LIN {X 0,Y 361.879,Z 141.036,A -85,B 0,C 180,E1 -13085.765,E2 -13085.765} C_VEL
LIN {X 0,Y 361.87,Z 141.034,A -85,B 0,C 180,E1 -13089.027,E2 -13089.027} C_VEL
LIN {X 0,Y 361.837,Z 141.037,A -85,B 0,C 180,E1 -13092.829,E2 -13092.829} C_VEL
LIN {X 0,Y 361.82,Z 141.044,A -85,B 0,C 180,E1 -13095.947,E2 -13095.947} C_VEL
LIN {X 0,Y 361.838,Z 141.042,A -85,B 0,C 180,E1 -13099.245,E2 -13099.245} C_VEL
LIN {X 0,Y 361.865,Z 141.033,A -85,B 0,C 180,E1 -13102.778,E2 -13102.778} C_VEL
LIN {X 0,Y 361.857,Z 141.036,A -85,B 0,C 180,E1 -13105.72,E2 -13105.72} C_VEL
LIN {X 0,Y 361.867,Z 141.03,A -85,B 0,C 180,E1 -13109.672,E2 -13109.672} C_VEL
LIN {X 0,Y 361.866,Z 141.018,A -85,B 0,C 180,E1 -13113.469,E2 -13113.469} C_VEL
LIN {X 0,Y 361.885,Z 141.028,A -85,B 0,C 180,E1 -13117.145,E2 -13117.145} C_VEL
LIN {X 0,Y 361.908,Z 141.031,A -85,B 0,C 180,E1 -13120.724,E2 -13120.724} C_VEL
LIN {X 0,Y 361.947,Z 141.019,A -85,B 0,C 180,E1 -13124.227,E2 -13124.227} C_VEL
LIN {X 0,Y 362.004,Z 141.017,A -85,B 0,C 180,E1 -13126.528,E2 -13126.528} C_VEL
LIN {X 0,Y 362.004,Z 141.016,A -85,B 0,C 180,E1 -13129.938,E2 -13129.938} C_VEL
LIN {X 0,Y 362.126,Z 140.997,A -85,B 0,C 180,E1 -13133.313,E2 -13133.313} C_VEL
LIN {X 0,Y 362.269,Z 140.97,A -85,B 0,C 180,E1 -13137.777,E2 -13137.777} C_VEL
LIN {X 0,Y 362.178,Z 140.979,A -85,B 0,C 180,E1 -13141.112,E2 -13141.112} C_VEL
LIN {X 0,Y 362.262,Z 140.976,A -85,B 0,C 180,E1 -13142.224,E2 -13142.224} C_VEL
LIN {X 0,Y 362.125,Z 140.992,A -85,B 0,C 180,E1 -13146.688,E2 -13146.688} C_VEL
LIN {X 0,Y 361.997,Z 140.99,A -85,B 0,C 180,E1 -13150.063,E2 -13150.063} C_VEL
LIN {X 0,Y 361.955,Z 141.024,A -85,B 0,C 180,E1 -13153.868,E2 -13153.868} C_VEL
LIN {X 0,Y 361.88,Z 141.031,A -85,B 0,C 180,E1 -13158.104,E2 -13158.104} C_VEL
LIN {X 0,Y 361.824,Z 141.034,A -85,B 0,C 180,E1 -13161.658,E2 -13161.658} C_VEL
LIN {X 0,Y 361.864,Z 141.037,A -85,B 0,C 180,E1 -13165.295,E2 -13165.295} C_VEL
LIN {X 0,Y 361.841,Z 141.012,A -85,B 0,C 180,E1 -13169.068,E2 -13169.068} C_VEL
LIN {X 0,Y 361.842,Z 141.028,A -85,B 0,C 180,E1 -13171.63,E2 -13171.63} C_VEL
LIN {X 0,Y 361.874,Z 141.028,A -85,B 0,C 180,E1 -13175.344,E2 -13175.344} C_VEL
LIN {X 0,Y 361.83,Z 141.018,A -85,B 0,C 180,E1 -13179.018,E2 -13179.018} C_VEL
LIN {X 0,Y 361.837,Z 141.039,A -85,B 0,C 180,E1 -13182.83,E2 -13182.83} C_VEL
LIN {X 0,Y 361.817,Z 141.02,A -85,B 0,C 180,E1 -13185.948,E2 -13185.948} C_VEL
LIN {X 0,Y 361.817,Z 141.04,A -85,B 0,C 180,E1 -13189.249,E2 -13189.249} C_VEL
LIN {X 0,Y 361.869,Z 141.025,A -85,B 0,C 180,E1 -13192.981,E2 -13192.981} C_VEL
LIN {X 0,Y 361.863,Z 141.027,A -85,B 0,C 180,E1 -13196.631,E2 -13196.631} C_VEL
LIN {X 0,Y 361.869,Z 141.035,A -85,B 0,C 180,E1 -13199.671,E2 -13199.671} C_VEL
LIN {X 0,Y 361.866,Z 141.036,A -85,B 0,C 180,E1 -13203.468,E2 -13203.468} C_VEL
LIN {X 0,Y 361.881,Z 141.033,A -85,B 0,C 180,E1 -13207.144,E2 -13207.144} C_VEL
LIN {X 0,Y 361.91,Z 141.025,A -85,B 0,C 180,E1 -13210.723,E2 -13210.723} C_VEL
LIN {X 0,Y 361.949,Z 141.027,A -85,B 0,C 180,E1 -13214.226,E2 -13214.226} C_VEL
LIN {X 0,Y 362.054,Z 141.133,A -85,B 0,C 180,E1 -13216.851,E2 -13216.851} C_VEL
LIN {X 0,Y 363.353,Z 146.545,A -85,B 0,C 180,E1 -13218.193,E2 -13218.193} C_VEL
LIN {X 0,Y 375.34,Z 174.664,A -85,B 0,C 180,E1 -13219.747,E2 -13219.747} C_VEL
LIN {X 0,Y 378.121,Z 181.605,A -85,B 0,C 180,E1 -13220.098,E2 -13220.098} C_VEL
LIN {X 0,Y 375.096,Z 311.282,A -85,B 0,C 180,E1 -13222.632,E2 -13222.632} C_VEL
LIN {X 0,Y 374.339,Z 326.412,A -85,B 0,C 180,E1 -13223.126,E2 -13223.126} C_VEL
LIN {X 0,Y 373.39,Z 340.483,A -85,B 0,C 180,E1 -13223.786,E2 -13223.786} C_VEL
LIN {X 0,Y 372.032,Z 355.504,A -85,B 0,C 180,E1 -13224.716,E2 -13224.716} C_VEL
LIN {X 0,Y 370.487,Z 370.541,A -85,B 0,C 180,E1 -13225.92,E2 -13225.92} C_VEL
LIN {X 0,Y 368.913,Z 383.973,A -85,B 0,C 180,E1 -13227.27,E2 -13227.27} C_VEL
LIN {X 0,Y 367.303,Z 396.209,A -85,B 0,C 180,E1 -13228.766,E2 -13228.766} C_VEL
LIN {X 0,Y 365.757,Z 407.68,A -85,B 0,C 180,E1 -13230.463,E2 -13230.463} C_VEL
LIN {X 0,Y 364.415,Z 417.514,A -85,B 0,C 180,E1 -13232.21,E2 -13232.21} C_VEL
LIN {X 0,Y 363.177,Z 426.655,A -85,B 0,C 180,E1 -13234.161,E2 -13234.161} C_VEL
LIN {X 0,Y 362.184,Z 434.264,A -85,B 0,C 180,E1 -13236.126,E2 -13236.126} C_VEL
LIN {X 0,Y 361.397,Z 441.384,A -85,B 0,C 180,E1 -13238.386,E2 -13238.386} C_VEL
LIN {X 0,Y 360.833,Z 447.004,A -85,B 0,C 180,E1 -13240.663,E2 -13240.663} C_VEL
LIN {X 0,Y 360.483,Z 451.14,A -85,B 0,C 180,E1 -13242.886,E2 -13242.886} C_VEL
LIN {X 0,Y 360.363,Z 452,A -85,B 0,C 180,E1 -13243.441,E2 -13243.441} C_VEL
LIN {X 0,Y 359.56,Z 453.289,A -85,B 0,C 180,E1 -13244.349,E2 -13244.349} C_VEL
LIN {X 0,Y 356.571,Z 454.897,A -85,B 0,C 180,E1 -13245.84,E2 -13245.84} C_VEL
LIN {X 0,Y 354.114,Z 455.843,A -85,B 0,C 180,E1 -13247.056,E2 -13247.056} C_VEL
LIN {X 0,Y 353.072,Z 456.303,A -85,B 0,C 180,E1 -13248.002,E2 -13248.002} C_VEL
LIN {X 0,Y 352.99,Z 456.411,A -85,B 0,C 180,E1 -13248.323,E2 -13248.323} C_VEL
LIN {X 0,Y 353.05,Z 456.561,A -85,B 0,C 180,E1 -13250.672,E2 -13250.672} C_VEL
LIN {X 0,Y 353.093,Z 456.028,A -85,B 0,C 180,E1 -13252.22,E2 -13252.22} C_VEL
LIN {X 0,Y 353.38,Z 454.051,A -85,B 0,C 180,E1 -13254.686,E2 -13254.686} C_VEL
LIN {X 0,Y 353.883,Z 450.673,A -85,B 0,C 180,E1 -13257.179,E2 -13257.179} C_VEL
LIN {X 0,Y 354.563,Z 445.772,A -85,B 0,C 180,E1 -13259.705,E2 -13259.705} C_VEL
LIN {X 0,Y 355.465,Z 440.501,A -85,B 0,C 180,E1 -13261.769,E2 -13261.769} C_VEL
LIN {X 0,Y 356.649,Z 433.956,A -85,B 0,C 180,E1 -13263.851,E2 -13263.851} C_VEL
LIN {X 0,Y 358.232,Z 425.446,A -85,B 0,C 180,E1 -13266.054,E2 -13266.054} C_VEL
LIN {X 0,Y 359.929,Z 416.53,A -85,B 0,C 180,E1 -13267.957,E2 -13267.957} C_VEL
LIN {X 0,Y 361.991,Z 405.841,A -85,B 0,C 180,E1 -13269.843,E2 -13269.843} C_VEL
LIN {X 0,Y 364.144,Z 394.025,A -85,B 0,C 180,E1 -13271.562,E2 -13271.562} C_VEL
LIN {X 0,Y 366.27,Z 381.307,A -85,B 0,C 180,E1 -13273.084,E2 -13273.084} C_VEL
LIN {X 0,Y 368.307,Z 368.431,A -85,B 0,C 180,E1 -13274.336,E2 -13274.336} C_VEL
LIN {X 0,Y 370.11,Z 354.336,A -85,B 0,C 180,E1 -13275.449,E2 -13275.449} C_VEL
LIN {X 0,Y 371.675,Z 340.065,A -85,B 0,C 180,E1 -13276.325,E2 -13276.325} C_VEL
LIN {X 0,Y 372.943,Z 325.224,A -85,B 0,C 180,E1 -13277.004,E2 -13277.004} C_VEL
LIN {X 0,Y 373.866,Z 310.283,A -85,B 0,C 180,E1 -13277.471,E2 -13277.471} C_VEL
LIN {X 0,Y 377.59,Z 188.012,A -85,B 0,C 180,E1 -13279.939,E2 -13279.939} C_VEL
LIN {X 0,Y 370.299,Z 172.503,A -85,B 0,C 180,E1 -13281.122,E2 -13281.122} C_VEL
LIN {X 0,Y 363.13,Z 159.246,A -85,B 0,C 180,E1 -13282.304,E2 -13282.304} C_VEL
LIN {X 0,Y 356.546,Z 147.757,A -85,B 0,C 180,E1 -13283.484,E2 -13283.484} C_VEL
LIN {X 0,Y 354.8,Z 141.906,A -85,B 0,C 180,E1 -13285.371,E2 -13285.371} C_VEL
LIN {X 0,Y 354.798,Z 141.908,A -85,B 0,C 180,E1 -13289.001,E2 -13289.001} C_VEL
LIN {X 0,Y 354.811,Z 141.899,A -85,B 0,C 180,E1 -13291.615,E2 -13291.615} C_VEL
LIN {X 0,Y 354.854,Z 141.892,A -85,B 0,C 180,E1 -13295.423,E2 -13295.423} C_VEL
LIN {X 0,Y 354.827,Z 141.91,A -85,B 0,C 180,E1 -13299.113,E2 -13299.113} C_VEL
LIN {X 0,Y 354.88,Z 141.902,A -85,B 0,C 180,E1 -13302.718,E2 -13302.718} C_VEL
LIN {X 0,Y 354.952,Z 141.897,A -85,B 0,C 180,E1 -13306.255,E2 -13306.255} C_VEL
LIN {X 0,Y 354.978,Z 141.894,A -85,B 0,C 180,E1 -13309.735,E2 -13309.735} C_VEL
LIN {X 0,Y 355.114,Z 141.874,A -85,B 0,C 180,E1 -13312.036,E2 -13312.036} C_VEL
LIN {X 0,Y 355.091,Z 141.87,A -85,B 0,C 180,E1 -13314.32,E2 -13314.32} C_VEL
LIN {X 0,Y 355.243,Z 141.853,A -85,B 0,C 180,E1 -13317.732,E2 -13317.732} C_VEL
LIN {X 0,Y 355.396,Z 141.84,A -85,B 0,C 180,E1 -13320,E2 -13320} C_VEL
LIN {X 0,Y 355.243,Z 141.855,A -85,B 0,C 180,E1 -13322.267,E2 -13322.267} C_VEL
LIN {X 0,Y 355.098,Z 141.877,A -85,B 0,C 180,E1 -13326.82,E2 -13326.82} C_VEL
LIN {X 0,Y 354.955,Z 141.893,A -85,B 0,C 180,E1 -13330.264,E2 -13330.264} C_VEL
LIN {X 0,Y 354.942,Z 141.896,A -85,B 0,C 180,E1 -13334.019,E2 -13334.019} C_VEL
LIN {X 0,Y 354.922,Z 141.899,A -85,B 0,C 180,E1 -13338.108,E2 -13338.108} C_VEL
LIN {X 0,Y 354.833,Z 141.909,A -85,B 0,C 180,E1 -13342.106,E2 -13342.106} C_VEL
LIN {X 0,Y 354.898,Z 141.898,A -85,B 0,C 180,E1 -13345.827,E2 -13345.827} C_VEL
LIN {X 0,Y 354.852,Z 141.903,A -85,B 0,C 180,E1 -13349.678,E2 -13349.678} C_VEL
LIN {X 0,Y 354.804,Z 141.914,A -85,B 0,C 180,E1 -13353.702,E2 -13353.702} C_VEL
LIN {X 0,Y 354.796,Z 141.917,A -85,B 0,C 180,E1 -13356.459,E2 -13356.459} C_VEL
LIN {X 0,Y 354.822,Z 141.896,A -85,B 0,C 180,E1 -13359.424,E2 -13359.424} C_VEL
LIN {X 0,Y 354.786,Z 141.901,A -85,B 0,C 180,E1 -13362.867,E2 -13362.867} C_VEL
LIN {X 0,Y 354.772,Z 141.909,A -85,B 0,C 180,E1 -13366.105,E2 -13366.105} C_VEL
LIN {X 0,Y 354.786,Z 141.911,A -85,B 0,C 180,E1 -13369.179,E2 -13369.179} C_VEL
LIN {X 0,Y 354.826,Z 141.959,A -85,B 0,C 180,E1 -13370.255,E2 -13370.255} C_VEL
LIN {X 0,Y 358.279,Z 153.223,A -85,B 0,C 180,E1 -13373.538,E2 -13373.538} C_VEL
LIN {X 0,Y 361.019,Z 163.125,A -85,B 0,C 180,E1 -13376.189,E2 -13376.189} C_VEL
LIN {X 0,Y 370.165,Z 181.186,A -85,B 0,C 180,E1 -13377.73,E2 -13377.73} C_VEL
LIN {X 0,Y 373.149,Z 188.13,A -85,B 0,C 180,E1 -13378.235,E2 -13378.235} C_VEL
LIN {X 0,Y 376.818,Z 207.275,A -85,B 0,C 180,E1 -13379.086,E2 -13379.086} C_VEL
LIN {X 0,Y 377.102,Z 209.697,A -85,B 0,C 180,E1 -13379.173,E2 -13379.173} C_VEL
LIN {X 0,Y 373.367,Z 329.597,A -85,B 0,C 180,E1 -13381.584,E2 -13381.584} C_VEL
LIN {X 0,Y 372.224,Z 345.584,A -85,B 0,C 180,E1 -13382.103,E2 -13382.103} C_VEL
LIN {X 0,Y 370.742,Z 360.136,A -85,B 0,C 180,E1 -13382.786,E2 -13382.786} C_VEL
LIN {X 0,Y 368.921,Z 374.936,A -85,B 0,C 180,E1 -13383.717,E2 -13383.717} C_VEL
LIN {X 0,Y 367.076,Z 388.167,A -85,B 0,C 180,E1 -13384.787,E2 -13384.787} C_VEL
LIN {X 0,Y 364.789,Z 401.788,A -85,B 0,C 180,E1 -13386.135,E2 -13386.135} C_VEL
LIN {X 0,Y 362.674,Z 414.145,A -85,B 0,C 180,E1 -13387.648,E2 -13387.648} C_VEL
LIN {X 0,Y 360.496,Z 425.702,A -85,B 0,C 180,E1 -13389.353,E2 -13389.353} C_VEL
LIN {X 0,Y 358.711,Z 435.703,A -85,B 0,C 180,E1 -13391.139,E2 -13391.139} C_VEL
LIN {X 0,Y 357.011,Z 444.998,A -85,B 0,C 180,E1 -13393.121,E2 -13393.121} C_VEL
LIN {X 0,Y 355.666,Z 452.763,A -85,B 0,C 180,E1 -13395.115,E2 -13395.115} C_VEL
LIN {X 0,Y 354.777,Z 458.414,A -85,B 0,C 180,E1 -13396.832,E2 -13396.832} C_VEL
LIN {X 0,Y 353.955,Z 464.549,A -85,B 0,C 180,E1 -13399.128,E2 -13399.128} C_VEL
LIN {X 0,Y 353.498,Z 469.304,A -85,B 0,C 180,E1 -13401.425,E2 -13401.425} C_VEL
LIN {X 0,Y 353.275,Z 473.279,A -85,B 0,C 180,E1 -13404.092,E2 -13404.092} C_VEL
LIN {X 0,Y 353.19,Z 475.51,A -85,B 0,C 180,E1 -13406.578,E2 -13406.578} C_VEL
LIN {X 0,Y 353.211,Z 476.343,A -85,B 0,C 180,E1 -13408.86,E2 -13408.86} C_VEL
LIN {X 0,Y 353.215,Z 476.037,A -85,B 0,C 180,E1 -13411.141,E2 -13411.141} C_VEL
LIN {X 0,Y 353.194,Z 474.577,A -85,B 0,C 180,E1 -13413.423,E2 -13413.423} C_VEL
LIN {X 0,Y 353.275,Z 471.617,A -85,B 0,C 180,E1 -13415.909,E2 -13415.909} C_VEL
LIN {X 0,Y 353.427,Z 467.984,A -85,B 0,C 180,E1 -13418.002,E2 -13418.002} C_VEL
LIN {X 0,Y 353.698,Z 462.674,A -85,B 0,C 180,E1 -13420.302,E2 -13420.302} C_VEL
LIN {X 0,Y 354.396,Z 455.88,A -85,B 0,C 180,E1 -13422.6,E2 -13422.6} C_VEL
LIN {X 0,Y 355.211,Z 448.529,A -85,B 0,C 180,E1 -13424.613,E2 -13424.613} C_VEL
LIN {X 0,Y 356.304,Z 439.69,A -85,B 0,C 180,E1 -13426.62,E2 -13426.62} C_VEL
LIN {X 0,Y 357.857,Z 429.042,A -85,B 0,C 180,E1 -13428.611,E2 -13428.611} C_VEL
LIN {X 0,Y 359.237,Z 418.762,A -85,B 0,C 180,E1 -13430.217,E2 -13430.217} C_VEL
LIN {X 0,Y 360.81,Z 407.288,A -85,B 0,C 180,E1 -13431.722,E2 -13431.722} C_VEL
LIN {X 0,Y 362.485,Z 394.416,A -85,B 0,C 180,E1 -13433.118,E2 -13433.118} C_VEL
LIN {X 0,Y 364.026,Z 382.022,A -85,B 0,C 180,E1 -13434.222,E2 -13434.222} C_VEL
LIN {X 0,Y 365.576,Z 367.655,A -85,B 0,C 180,E1 -13435.248,E2 -13435.248} C_VEL
LIN {X 0,Y 366.71,Z 353.667,A -85,B 0,C 180,E1 -13436.031,E2 -13436.031} C_VEL
LIN {X 0,Y 367.849,Z 338.418,A -85,B 0,C 180,E1 -13436.641,E2 -13436.641} C_VEL
LIN {X 0,Y 368.459,Z 322.812,A -85,B 0,C 180,E1 -13437.052,E2 -13437.052} C_VEL
LIN {X 0,Y 371.276,Z 207.418,A -85,B 0,C 180,E1 -13439.317,E2 -13439.317} C_VEL
LIN {X 0,Y 365.889,Z 177.835,A -85,B 0,C 180,E1 -13440.363,E2 -13440.363} C_VEL
LIN {X 0,Y 360.228,Z 163.937,A -85,B 0,C 180,E1 -13441.146,E2 -13441.146} C_VEL
LIN {X 0,Y 356.983,Z 150.277,A -85,B 0,C 180,E1 -13444.223,E2 -13444.223} C_VEL
LIN {X 0,Y 354.838,Z 141.912,A -85,B 0,C 180,E1 -13446.245,E2 -13446.245} C_VEL
LIN {X 0,Y 354.825,Z 141.914,A -85,B 0,C 180,E1 -13449.424,E2 -13449.424} C_VEL
LIN {X 0,Y 354.789,Z 141.916,A -85,B 0,C 180,E1 -13452.868,E2 -13452.868} C_VEL
LIN {X 0,Y 354.769,Z 141.922,A -85,B 0,C 180,E1 -13456.104,E2 -13456.104} C_VEL
LIN {X 0,Y 354.79,Z 141.921,A -85,B 0,C 180,E1 -13459.18,E2 -13459.18} C_VEL
LIN {X 0,Y 354.808,Z 141.911,A -85,B 0,C 180,E1 -13462.403,E2 -13462.403} C_VEL
LIN {X 0,Y 354.814,Z 141.911,A -85,B 0,C 180,E1 -13464.941,E2 -13464.941} C_VEL
LIN {X 0,Y 354.796,Z 141.913,A -85,B 0,C 180,E1 -13468.406,E2 -13468.406} C_VEL
LIN {X 0,Y 354.802,Z 141.894,A -85,B 0,C 180,E1 -13471.615,E2 -13471.615} C_VEL
LIN {X 0,Y 354.838,Z 141.907,A -85,B 0,C 180,E1 -13475.658,E2 -13475.658} C_VEL
LIN {X 0,Y 354.83,Z 141.907,A -85,B 0,C 180,E1 -13479.114,E2 -13479.114} C_VEL
LIN {X 0,Y 354.884,Z 141.898,A -85,B 0,C 180,E1 -13482.72,E2 -13482.72} C_VEL
LIN {X 0,Y 354.956,Z 141.896,A -85,B 0,C 180,E1 -13486.256,E2 -13486.256} C_VEL
LIN {X 0,Y 354.96,Z 141.892,A -85,B 0,C 180,E1 -13489.736,E2 -13489.736} C_VEL
LIN {X 0,Y 355.092,Z 141.874,A -85,B 0,C 180,E1 -13493.18,E2 -13493.18} C_VEL
LIN {X 0,Y 355.231,Z 141.847,A -85,B 0,C 180,E1 -13497.733,E2 -13497.733} C_VEL
LIN {X 0,Y 355.149,Z 141.854,A -85,B 0,C 180,E1 -13501.134,E2 -13501.134} C_VEL
LIN {X 0,Y 355.224,Z 141.853,A -85,B 0,C 180,E1 -13502.268,E2 -13502.268} C_VEL
LIN {X 0,Y 355.092,Z 141.867,A -85,B 0,C 180,E1 -13506.821,E2 -13506.821} C_VEL
LIN {X 0,Y 354.953,Z 141.868,A -85,B 0,C 180,E1 -13510.265,E2 -13510.265} C_VEL
LIN {X 0,Y 354.897,Z 141.903,A -85,B 0,C 180,E1 -13513.986,E2 -13513.986} C_VEL
LIN {X 0,Y 354.837,Z 141.908,A -85,B 0,C 180,E1 -13518.064,E2 -13518.064} C_VEL
LIN {X 0,Y 354.791,Z 141.909,A -85,B 0,C 180,E1 -13522.109,E2 -13522.109} C_VEL
LIN {X 0,Y 354.803,Z 141.91,A -85,B 0,C 180,E1 -13525.836,E2 -13525.836} C_VEL
LIN {X 0,Y 354.79,Z 141.889,A -85,B 0,C 180,E1 -13529.685,E2 -13529.685} C_VEL
LIN {X 0,Y 354.791,Z 141.908,A -85,B 0,C 180,E1 -13532.334,E2 -13532.334} C_VEL
LIN {X 0,Y 354.823,Z 141.904,A -85,B 0,C 180,E1 -13535.698,E2 -13535.698} C_VEL
LIN {X 0,Y 354.773,Z 141.901,A -85,B 0,C 180,E1 -13539.413,E2 -13539.413} C_VEL
LIN {X 0,Y 354.789,Z 141.916,A -85,B 0,C 180,E1 -13542.866,E2 -13542.866} C_VEL
LIN {X 0,Y 354.767,Z 141.898,A -85,B 0,C 180,E1 -13546.103,E2 -13546.103} C_VEL
LIN {X 0,Y 354.77,Z 141.918,A -85,B 0,C 180,E1 -13549.176,E2 -13549.176} C_VEL
LIN {X 0,Y 354.805,Z 141.901,A -85,B 0,C 180,E1 -13552.404,E2 -13552.404} C_VEL
LIN {X 0,Y 354.816,Z 141.913,A -85,B 0,C 180,E1 -13554.941,E2 -13554.941} C_VEL
LIN {X 0,Y 354.798,Z 141.91,A -85,B 0,C 180,E1 -13558.405,E2 -13558.405} C_VEL
LIN {X 0,Y 354.804,Z 141.909,A -85,B 0,C 180,E1 -13561.614,E2 -13561.614} C_VEL
LIN {X 0,Y 354.811,Z 141.915,A -85,B 0,C 180,E1 -13565.419,E2 -13565.419} C_VEL
LIN {X 0,Y 354.832,Z 141.91,A -85,B 0,C 180,E1 -13569.113,E2 -13569.113} C_VEL
LIN {X 0,Y 354.885,Z 141.887,A -85,B 0,C 180,E1 -13572.719,E2 -13572.719} C_VEL
LIN {X 0,Y 355,Z 142.038,A -85,B 0,C 180,E1 -13576.402,E2 -13576.402} C_VEL
LIN {X 0,Y 356.226,Z 147.086,A -85,B 0,C 180,E1 -13577.637,E2 -13577.637} C_VEL
LIN {X 0,Y 368.488,Z 175.376,A -85,B 0,C 180,E1 -13579.247,E2 -13579.247} C_VEL
LIN {X 0,Y 371.75,Z 183.518,A -85,B 0,C 180,E1 -13579.668,E2 -13579.668} C_VEL
LIN {X 0,Y 368.535,Z 312.21,A -85,B 0,C 180,E1 -13582.225,E2 -13582.225} C_VEL
LIN {X 0,Y 367.701,Z 327.89,A -85,B 0,C 180,E1 -13582.759,E2 -13582.759} C_VEL
LIN {X 0,Y 366.687,Z 342.3,A -85,B 0,C 180,E1 -13583.465,E2 -13583.465} C_VEL
LIN {X 0,Y 365.379,Z 355.987,A -85,B 0,C 180,E1 -13584.342,E2 -13584.342} C_VEL
LIN {X 0,Y 363.97,Z 369.407,A -85,B 0,C 180,E1 -13585.431,E2 -13585.431} C_VEL
LIN {X 0,Y 362.295,Z 383.114,A -85,B 0,C 180,E1 -13586.802,E2 -13586.802} C_VEL
LIN {X 0,Y 360.596,Z 395.529,A -85,B 0,C 180,E1 -13588.324,E2 -13588.324} C_VEL
LIN {X 0,Y 359.028,Z 406.818,A -85,B 0,C 180,E1 -13590,E2 -13590} C_VEL
LIN {X 0,Y 357.709,Z 416.331,A -85,B 0,C 180,E1 -13591.688,E2 -13591.688} C_VEL
LIN {X 0,Y 356.366,Z 425.713,A -85,B 0,C 180,E1 -13593.674,E2 -13593.674} C_VEL
LIN {X 0,Y 355.302,Z 433.529,A -85,B 0,C 180,E1 -13595.675,E2 -13595.675} C_VEL
LIN {X 0,Y 354.452,Z 440.836,A -85,B 0,C 180,E1 -13597.978,E2 -13597.978} C_VEL
LIN {X 0,Y 353.797,Z 446.631,A -85,B 0,C 180,E1 -13600.298,E2 -13600.298} C_VEL
LIN {X 0,Y 353.438,Z 451.033,A -85,B 0,C 180,E1 -13602.634,E2 -13602.634} C_VEL
LIN {X 0,Y 353.107,Z 454.159,A -85,B 0,C 180,E1 -13604.995,E2 -13604.995} C_VEL
LIN {X 0,Y 353.039,Z 456.034,A -85,B 0,C 180,E1 -13607.374,E2 -13607.374} C_VEL
LIN {X 0,Y 352.99,Z 456.411,A -85,B 0,C 180,E1 -13608.323,E2 -13608.323} C_VEL
LIN {X 0,Y 352.321,Z 456.687,A -85,B 0,C 180,E1 -13609.275,E2 -13609.275} C_VEL
LIN {X 0,Y 349.461,Z 456.693,A -85,B 0,C 180,E1 -13610.826,E2 -13610.826} C_VEL
LIN {X 0,Y 347.091,Z 456.3,A -85,B 0,C 180,E1 -13612.081,E2 -13612.081} C_VEL
LIN {X 0,Y 346.146,Z 455.783,A -85,B 0,C 180,E1 -13613.048,E2 -13613.048} C_VEL
LIN {X 0,Y 346.108,Z 455.534,A -85,B 0,C 180,E1 -13613.374,E2 -13613.374} C_VEL
LIN {X 0,Y 346.372,Z 453.872,A -85,B 0,C 180,E1 -13615.22,E2 -13615.22} C_VEL
LIN {X 0,Y 346.917,Z 450.294,A -85,B 0,C 180,E1 -13617.771,E2 -13617.771} C_VEL
LIN {X 0,Y 347.737,Z 445.156,A -85,B 0,C 180,E1 -13620.349,E2 -13620.349} C_VEL
LIN {X 0,Y 348.765,Z 439.682,A -85,B 0,C 180,E1 -13622.477,E2 -13622.477} C_VEL
LIN {X 0,Y 350.086,Z 432.868,A -85,B 0,C 180,E1 -13624.605,E2 -13624.605} C_VEL
LIN {X 0,Y 351.867,Z 424.207,A -85,B 0,C 180,E1 -13626.813,E2 -13626.813} C_VEL
LIN {X 0,Y 353.658,Z 414.975,A -85,B 0,C 180,E1 -13628.754,E2 -13628.754} C_VEL
LIN {X 0,Y 355.894,Z 403.932,A -85,B 0,C 180,E1 -13630.667,E2 -13630.667} C_VEL
LIN {X 0,Y 358.205,Z 391.69,A -85,B 0,C 180,E1 -13632.41,E2 -13632.41} C_VEL
LIN {X 0,Y 360.301,Z 379.771,A -85,B 0,C 180,E1 -13633.803,E2 -13633.803} C_VEL
LIN {X 0,Y 362.397,Z 366.663,A -85,B 0,C 180,E1 -13635.06,E2 -13635.06} C_VEL
LIN {X 0,Y 364.223,Z 352.726,A -85,B 0,C 180,E1 -13636.142,E2 -13636.142} C_VEL
LIN {X 0,Y 365.803,Z 338.606,A -85,B 0,C 180,E1 -13636.991,E2 -13636.991} C_VEL
LIN {X 0,Y 367.041,Z 324.609,A -85,B 0,C 180,E1 -13637.62,E2 -13637.62} C_VEL
LIN {X 0,Y 367.904,Z 310.5,A -85,B 0,C 180,E1 -13638.066,E2 -13638.066} C_VEL
LIN {X 0,Y 371.748,Z 190.159,A -85,B 0,C 180,E1 -13640.529,E2 -13640.529} C_VEL
LIN {X 0,Y 364.564,Z 175.02,A -85,B 0,C 180,E1 -13641.734,E2 -13641.734} C_VEL
LIN {X 0,Y 356.643,Z 160.458,A -85,B 0,C 180,E1 -13643.1,E2 -13643.1} C_VEL
LIN {X 0,Y 351.183,Z 151.357,A -85,B 0,C 180,E1 -13644.077,E2 -13644.077} C_VEL
LIN {X 0,Y 349.378,Z 148.082,A -85,B 0,C 180,E1 -13644.445,E2 -13644.445} C_VEL
LIN {X 0,Y 347.773,Z 142.789,A -85,B 0,C 180,E1 -13646.234,E2 -13646.234} C_VEL
LIN {X 0,Y 347.745,Z 142.795,A -85,B 0,C 180,E1 -13649.651,E2 -13649.651} C_VEL
LIN {X 0,Y 347.785,Z 142.789,A -85,B 0,C 180,E1 -13653.603,E2 -13653.603} C_VEL
LIN {X 0,Y 347.784,Z 142.77,A -85,B 0,C 180,E1 -13656.161,E2 -13656.161} C_VEL
LIN {X 0,Y 347.806,Z 142.783,A -85,B 0,C 180,E1 -13659.908,E2 -13659.908} C_VEL
LIN {X 0,Y 347.832,Z 142.784,A -85,B 0,C 180,E1 -13663.568,E2 -13663.568} C_VEL
LIN {X 0,Y 347.89,Z 142.775,A -85,B 0,C 180,E1 -13667.16,E2 -13667.16} C_VEL
LIN {X 0,Y 348.094,Z 142.745,A -85,B 0,C 180,E1 -13671.612,E2 -13671.612} C_VEL
LIN {X 0,Y 348.066,Z 142.746,A -85,B 0,C 180,E1 -13674.205,E2 -13674.205} C_VEL
LIN {X 0,Y 348.205,Z 142.729,A -85,B 0,C 180,E1 -13677.686,E2 -13677.686} C_VEL
LIN {X 0,Y 348.345,Z 142.718,A -85,B 0,C 180,E1 -13680,E2 -13680} C_VEL
LIN {X 0,Y 348.206,Z 142.732,A -85,B 0,C 180,E1 -13682.313,E2 -13682.313} C_VEL
LIN {X 0,Y 348.063,Z 142.754,A -85,B 0,C 180,E1 -13686.958,E2 -13686.958} C_VEL
LIN {X 0,Y 347.896,Z 142.774,A -85,B 0,C 180,E1 -13690.475,E2 -13690.475} C_VEL
LIN {X 0,Y 347.897,Z 142.773,A -85,B 0,C 180,E1 -13694.149,E2 -13694.149} C_VEL
LIN {X 0,Y 347.89,Z 142.775,A -85,B 0,C 180,E1 -13698.29,E2 -13698.29} C_VEL
LIN {X 0,Y 347.787,Z 142.787,A -85,B 0,C 180,E1 -13701.635,E2 -13701.635} C_VEL
LIN {X 0,Y 347.811,Z 142.784,A -85,B 0,C 180,E1 -13705.108,E2 -13705.108} C_VEL
LIN {X 0,Y 347.809,Z 142.785,A -85,B 0,C 180,E1 -13707.694,E2 -13707.694} C_VEL
LIN {X 0,Y 347.762,Z 142.79,A -85,B 0,C 180,E1 -13710.346,E2 -13710.346} C_VEL
LIN {X 0,Y 347.742,Z 142.791,A -85,B 0,C 180,E1 -13714.464,E2 -13714.464} C_VEL
LIN {X 0,Y 347.771,Z 142.774,A -85,B 0,C 180,E1 -13717.988,E2 -13717.988} C_VEL
LIN {X 0,Y 347.748,Z 142.787,A -85,B 0,C 180,E1 -13721.83,E2 -13721.83} C_VEL
LIN {X 0,Y 347.764,Z 142.793,A -85,B 0,C 180,E1 -13725.017,E2 -13725.017} C_VEL
LIN {X 0,Y 347.761,Z 142.789,A -85,B 0,C 180,E1 -13728.944,E2 -13728.944} C_VEL
LIN {X 0,Y 347.761,Z 142.903,A -85,B 0,C 180,E1 -13729.391,E2 -13729.391} C_VEL
LIN {X 0,Y 351.251,Z 154.011,A -85,B 0,C 180,E1 -13732.774,E2 -13732.774} C_VEL
LIN {X 0,Y 353.862,Z 163.089,A -85,B 0,C 180,E1 -13735.258,E2 -13735.258} C_VEL
LIN {X 0,Y 363.123,Z 180.892,A -85,B 0,C 180,E1 -13736.895,E2 -13736.895} C_VEL
LIN {X 0,Y 367.729,Z 191.04,A -85,B 0,C 180,E1 -13737.69,E2 -13737.69} C_VEL
LIN {X 0,Y 371.148,Z 209.403,A -85,B 0,C 180,E1 -13738.521,E2 -13738.521} C_VEL
LIN {X 0,Y 369.725,Z 257.449,A -85,B 0,C 180,E1 -13739.508,E2 -13739.508} C_VEL
LIN {X 0,Y 367.386,Z 329.786,A -85,B 0,C 180,E1 -13741,E2 -13741} C_VEL
LIN {X 0,Y 366.183,Z 345.589,A -85,B 0,C 180,E1 -13741.523,E2 -13741.523} C_VEL
LIN {X 0,Y 364.64,Z 360.075,A -85,B 0,C 180,E1 -13742.213,E2 -13742.213} C_VEL
LIN {X 0,Y 362.755,Z 374.729,A -85,B 0,C 180,E1 -13743.15,E2 -13743.15} C_VEL
LIN {X 0,Y 360.706,Z 388.806,A -85,B 0,C 180,E1 -13744.309,E2 -13744.309} C_VEL
LIN {X 0,Y 358.333,Z 402.268,A -85,B 0,C 180,E1 -13745.678,E2 -13745.678} C_VEL
LIN {X 0,Y 355.919,Z 415.512,A -85,B 0,C 180,E1 -13747.354,E2 -13747.354} C_VEL
LIN {X 0,Y 353.728,Z 426.576,A -85,B 0,C 180,E1 -13749.046,E2 -13749.046} C_VEL
LIN {X 0,Y 351.695,Z 437.341,A -85,B 0,C 180,E1 -13751.051,E2 -13751.051} C_VEL
LIN {X 0,Y 349.963,Z 446.338,A -85,B 0,C 180,E1 -13753.071,E2 -13753.071} C_VEL
LIN {X 0,Y 348.371,Z 454.744,A -85,B 0,C 180,E1 -13755.374,E2 -13755.374} C_VEL
LIN {X 0,Y 347.399,Z 461.649,A -85,B 0,C 180,E1 -13757.736,E2 -13757.736} C_VEL
LIN {X 0,Y 346.643,Z 467.04,A -85,B 0,C 180,E1 -13760.077,E2 -13760.077} C_VEL
LIN {X 0,Y 346.366,Z 470.203,A -85,B 0,C 180,E1 -13761.835,E2 -13761.835} C_VEL
LIN {X 0,Y 346.158,Z 473.387,A -85,B 0,C 180,E1 -13764.174,E2 -13764.174} C_VEL
LIN {X 0,Y 346.112,Z 475.359,A -85,B 0,C 180,E1 -13766.508,E2 -13766.508} C_VEL
LIN {X 0,Y 346.111,Z 476.152,A -85,B 0,C 180,E1 -13768.837,E2 -13768.837} C_VEL
LIN {X 0,Y 346.115,Z 475.808,A -85,B 0,C 180,E1 -13771.164,E2 -13771.164} C_VEL
LIN {X 0,Y 346.117,Z 474.31,A -85,B 0,C 180,E1 -13773.493,E2 -13773.493} C_VEL
LIN {X 0,Y 346.195,Z 471.531,A -85,B 0,C 180,E1 -13775.885,E2 -13775.885} C_VEL
LIN {X 0,Y 346.35,Z 467.651,A -85,B 0,C 180,E1 -13778.166,E2 -13778.166} C_VEL
LIN {X 0,Y 346.656,Z 462.293,A -85,B 0,C 180,E1 -13780.514,E2 -13780.514} C_VEL
LIN {X 0,Y 347.398,Z 455.448,A -85,B 0,C 180,E1 -13782.858,E2 -13782.858} C_VEL
LIN {X 0,Y 348.245,Z 448.159,A -85,B 0,C 180,E1 -13784.881,E2 -13784.881} C_VEL
LIN {X 0,Y 349.422,Z 439.141,A -85,B 0,C 180,E1 -13786.957,E2 -13786.957} C_VEL
LIN {X 0,Y 351.044,Z 428.421,A -85,B 0,C 180,E1 -13788.986,E2 -13788.986} C_VEL
LIN {X 0,Y 352.574,Z 416.976,A -85,B 0,C 180,E1 -13790.782,E2 -13790.782} C_VEL
LIN {X 0,Y 354.32,Z 405.291,A -85,B 0,C 180,E1 -13792.294,E2 -13792.294} C_VEL
LIN {X 0,Y 356.03,Z 392.025,A -85,B 0,C 180,E1 -13793.716,E2 -13793.716} C_VEL
LIN {X 0,Y 357.701,Z 379.124,A -85,B 0,C 180,E1 -13794.833,E2 -13794.833} C_VEL
LIN {X 0,Y 359.238,Z 364.426,A -85,B 0,C 180,E1 -13795.852,E2 -13795.852} C_VEL
LIN {X 0,Y 360.493,Z 349.412,A -85,B 0,C 180,E1 -13796.642,E2 -13796.642} C_VEL
LIN {X 0,Y 361.522,Z 333.568,A -85,B 0,C 180,E1 -13797.223,E2 -13797.223} C_VEL
LIN {X 0,Y 362.268,Z 311.772,A -85,B 0,C 180,E1 -13797.71,E2 -13797.71} C_VEL
LIN {X 0,Y 364.858,Z 208.371,A -85,B 0,C 180,E1 -13799.773,E2 -13799.773} C_VEL
LIN {X 0,Y 359.888,Z 180.715,A -85,B 0,C 180,E1 -13800.769,E2 -13800.769} C_VEL
LIN {X 0,Y 352.97,Z 163.804,A -85,B 0,C 180,E1 -13801.733,E2 -13801.733} C_VEL
LIN {X 0,Y 349.987,Z 151.467,A -85,B 0,C 180,E1 -13804.583,E2 -13804.583} C_VEL
LIN {X 0,Y 347.786,Z 142.793,A -85,B 0,C 180,E1 -13806.698,E2 -13806.698} C_VEL
LIN {X 0,Y 347.733,Z 142.797,A -85,B 0,C 180,E1 -13810.298,E2 -13810.298} C_VEL
LIN {X 0,Y 347.724,Z 142.8,A -85,B 0,C 180,E1 -13813.409,E2 -13813.409} C_VEL
LIN {X 0,Y 347.727,Z 142.799,A -85,B 0,C 180,E1 -13816.687,E2 -13816.687} C_VEL
LIN {X 0,Y 347.749,Z 142.788,A -85,B 0,C 180,E1 -13820.174,E2 -13820.174} C_VEL
LIN {X 0,Y 347.763,Z 142.789,A -85,B 0,C 180,E1 -13822.68,E2 -13822.68} C_VEL
LIN {X 0,Y 347.751,Z 142.792,A -85,B 0,C 180,E1 -13825.957,E2 -13825.957} C_VEL
LIN {X 0,Y 347.743,Z 142.79,A -85,B 0,C 180,E1 -13829.652,E2 -13829.652} C_VEL
LIN {X 0,Y 347.752,Z 142.777,A -85,B 0,C 180,E1 -13833.602,E2 -13833.602} C_VEL
LIN {X 0,Y 347.778,Z 142.786,A -85,B 0,C 180,E1 -13836.162,E2 -13836.162} C_VEL
LIN {X 0,Y 347.809,Z 142.782,A -85,B 0,C 180,E1 -13839.91,E2 -13839.91} C_VEL
LIN {X 0,Y 347.836,Z 142.775,A -85,B 0,C 180,E1 -13843.569,E2 -13843.569} C_VEL
LIN {X 0,Y 347.894,Z 142.768,A -85,B 0,C 180,E1 -13847.161,E2 -13847.161} C_VEL
LIN {X 0,Y 347.939,Z 142.768,A -85,B 0,C 180,E1 -13850.701,E2 -13850.701} C_VEL
LIN {X 0,Y 348.043,Z 142.756,A -85,B 0,C 180,E1 -13854.206,E2 -13854.206} C_VEL
LIN {X 0,Y 348.192,Z 142.723,A -85,B 0,C 180,E1 -13857.687,E2 -13857.687} C_VEL
LIN {X 0,Y 348.121,Z 142.729,A -85,B 0,C 180,E1 -13861.157,E2 -13861.157} C_VEL
LIN {X 0,Y 348.185,Z 142.73,A -85,B 0,C 180,E1 -13862.314,E2 -13862.314} C_VEL
LIN {X 0,Y 348.059,Z 142.743,A -85,B 0,C 180,E1 -13866.959,E2 -13866.959} C_VEL
LIN {X 0,Y 347.892,Z 142.749,A -85,B 0,C 180,E1 -13870.476,E2 -13870.476} C_VEL
LIN {X 0,Y 347.856,Z 142.779,A -85,B 0,C 180,E1 -13874.119,E2 -13874.119} C_VEL
LIN {X 0,Y 347.79,Z 142.785,A -85,B 0,C 180,E1 -13878.237,E2 -13878.237} C_VEL
LIN {X 0,Y 347.748,Z 142.787,A -85,B 0,C 180,E1 -13881.616,E2 -13881.616} C_VEL
LIN {X 0,Y 347.741,Z 142.795,A -85,B 0,C 180,E1 -13885.114,E2 -13885.114} C_VEL
LIN {X 0,Y 347.729,Z 142.778,A -85,B 0,C 180,E1 -13887.702,E2 -13887.702} C_VEL
LIN {X 0,Y 347.737,Z 142.771,A -85,B 0,C 180,E1 -13890.35,E2 -13890.35} C_VEL
LIN {X 0,Y 347.753,Z 142.79,A -85,B 0,C 180,E1 -13894.044,E2 -13894.044} C_VEL
LIN {X 0,Y 347.759,Z 142.769,A -85,B 0,C 180,E1 -13897.322,E2 -13897.322} C_VEL
LIN {X 0,Y 347.746,Z 142.791,A -85,B 0,C 180,E1 -13901.601,E2 -13901.601} C_VEL
LIN {X 0,Y 347.704,Z 142.78,A -85,B 0,C 180,E1 -13905.028,E2 -13905.028} C_VEL
LIN {X 0,Y 347.746,Z 142.791,A -85,B 0,C 180,E1 -13908.399,E2 -13908.399} C_VEL
LIN {X 0,Y 347.761,Z 142.779,A -85,B 0,C 180,E1 -13912.678,E2 -13912.678} C_VEL
LIN {X 0,Y 347.754,Z 142.792,A -85,B 0,C 180,E1 -13915.956,E2 -13915.956} C_VEL
LIN {X 0,Y 347.746,Z 142.794,A -85,B 0,C 180,E1 -13919.651,E2 -13919.651} C_VEL
LIN {X 0,Y 347.749,Z 142.796,A -85,B 0,C 180,E1 -13923.6,E2 -13923.6} C_VEL
LIN {X 0,Y 347.757,Z 142.795,A -85,B 0,C 180,E1 -13926.159,E2 -13926.159} C_VEL
LIN {X 0,Y 347.811,Z 142.788,A -85,B 0,C 180,E1 -13929.909,E2 -13929.909} C_VEL
LIN {X 0,Y 347.837,Z 142.773,A -85,B 0,C 180,E1 -13933.568,E2 -13933.568} C_VEL
LIN {X 0,Y 347.909,Z 142.796,A -85,B 0,C 180,E1 -13935.906,E2 -13935.906} C_VEL
LIN {X 0,Y 348.94,Z 147.03,A -85,B 0,C 180,E1 -13937.005,E2 -13937.005} C_VEL
LIN {X 0,Y 361.391,Z 175.438,A -85,B 0,C 180,E1 -13938.697,E2 -13938.697} C_VEL
LIN {X 0,Y 365.326,Z 185.606,A -85,B 0,C 180,E1 -13939.229,E2 -13939.229} C_VEL
LIN {X 0,Y 362.066,Z 311.741,A -85,B 0,C 180,E1 -13941.769,E2 -13941.769} C_VEL
LIN {X 0,Y 361.201,Z 327.692,A -85,B 0,C 180,E1 -13942.312,E2 -13942.312} C_VEL
LIN {X 0,Y 360.19,Z 341.575,A -85,B 0,C 180,E1 -13942.995,E2 -13942.995} C_VEL
LIN {X 0,Y 358.756,Z 356.439,A -85,B 0,C 180,E1 -13943.955,E2 -13943.955} C_VEL
LIN {X 0,Y 357.287,Z 369.828,A -85,B 0,C 180,E1 -13945.063,E2 -13945.063} C_VEL
LIN {X 0,Y 355.682,Z 382.228,A -85,B 0,C 180,E1 -13946.318,E2 -13946.318} C_VEL
LIN {X 0,Y 353.933,Z 394.821,A -85,B 0,C 180,E1 -13947.866,E2 -13947.866} C_VEL
LIN {X 0,Y 352.415,Z 405.37,A -85,B 0,C 180,E1 -13949.428,E2 -13949.428} C_VEL
LIN {X 0,Y 351.025,Z 415.15,A -85,B 0,C 180,E1 -13951.147,E2 -13951.147} C_VEL
LIN {X 0,Y 349.542,Z 424.776,A -85,B 0,C 180,E1 -13953.169,E2 -13953.169} C_VEL
LIN {X 0,Y 348.45,Z 432.785,A -85,B 0,C 180,E1 -13955.207,E2 -13955.207} C_VEL
LIN {X 0,Y 347.564,Z 439.958,A -85,B 0,C 180,E1 -13957.438,E2 -13957.438} C_VEL
LIN {X 0,Y 346.79,Z 446.245,A -85,B 0,C 180,E1 -13959.919,E2 -13959.919} C_VEL
LIN {X 0,Y 346.494,Z 449.78,A -85,B 0,C 180,E1 -13961.702,E2 -13961.702} C_VEL
LIN {X 0,Y 346.083,Z 453.362,A -85,B 0,C 180,E1 -13964.104,E2 -13964.104} C_VEL
LIN {X 0,Y 345.963,Z 455.676,A -85,B 0,C 180,E1 -13966.523,E2 -13966.523} C_VEL
LIN {X 0,Y 345.912,Z 456.76,A -85,B 0,C 180,E1 -13968.97,E2 -13968.97} C_VEL
LIN {X 0,Y 345.99,Z 456.588,A -85,B 0,C 180,E1 -13971.446,E2 -13971.446} C_VEL
LIN {X 0,Y 346.108,Z 455.534,A -85,B 0,C 180,E1 -13973.374,E2 -13973.374} C_VEL
LIN {X 0,Y 345.584,Z 454.8,A -85,B 0,C 180,E1 -13974.34,E2 -13974.34} C_VEL
LIN {X 0,Y 342.973,Z 453.295,A -85,B 0,C 180,E1 -13975.912,E2 -13975.912} C_VEL
LIN {X 0,Y 340.805,Z 451.749,A -85,B 0,C 180,E1 -13977.173,E2 -13977.173} C_VEL
LIN {X 0,Y 340.008,Z 450.319,A -85,B 0,C 180,E1 -13978.133,E2 -13978.133} C_VEL
LIN {X 0,Y 340.018,Z 449.76,A -85,B 0,C 180,E1 -13978.454,E2 -13978.454} C_VEL
LIN {X 0,Y 340.965,Z 444.533,A -85,B 0,C 180,E1 -13981.017,E2 -13981.017} C_VEL
LIN {X 0,Y 342.008,Z 439.333,A -85,B 0,C 180,E1 -13983.025,E2 -13983.025} C_VEL
LIN {X 0,Y 343.311,Z 432.995,A -85,B 0,C 180,E1 -13985.029,E2 -13985.029} C_VEL
LIN {X 0,Y 345.132,Z 424.576,A -85,B 0,C 180,E1 -13987.215,E2 -13987.215} C_VEL
LIN {X 0,Y 347.054,Z 415.333,A -85,B 0,C 180,E1 -13989.197,E2 -13989.197} C_VEL
LIN {X 0,Y 349.461,Z 404.008,A -85,B 0,C 180,E1 -13991.195,E2 -13991.195} C_VEL
LIN {X 0,Y 351.89,Z 391.768,A -85,B 0,C 180,E1 -13992.964,E2 -13992.964} C_VEL
LIN {X 0,Y 354.356,Z 378.481,A -85,B 0,C 180,E1 -13994.525,E2 -13994.525} C_VEL
LIN {X 0,Y 356.559,Z 364.986,A -85,B 0,C 180,E1 -13995.805,E2 -13995.805} C_VEL
LIN {X 0,Y 358.529,Z 350.47,A -85,B 0,C 180,E1 -13996.902,E2 -13996.902} C_VEL
LIN {X 0,Y 360.164,Z 335.258,A -85,B 0,C 180,E1 -13997.781,E2 -13997.781} C_VEL
LIN {X 0,Y 361.472,Z 320.023,A -85,B 0,C 180,E1 -13998.408,E2 -13998.408} C_VEL
LIN {X 0,Y 362.213,Z 303.969,A -85,B 0,C 180,E1 -13998.844,E2 -13998.844} C_VEL
LIN {X 0,Y 366.033,Z 192.592,A -85,B 0,C 180,E1 -14001.125,E2 -14001.125} C_VEL
LIN {X 0,Y 359.817,Z 179.396,A -85,B 0,C 180,E1 -14002.205,E2 -14002.205} C_VEL
LIN {X 0,Y 352.216,Z 165.217,A -85,B 0,C 180,E1 -14003.563,E2 -14003.563} C_VEL
LIN {X 0,Y 344.683,Z 152.622,A -85,B 0,C 180,E1 -14004.963,E2 -14004.963} C_VEL
LIN {X 0,Y 342.126,Z 148.361,A -85,B 0,C 180,E1 -14005.487,E2 -14005.487} C_VEL
LIN {X 0,Y 340.704,Z 143.664,A -85,B 0,C 180,E1 -14007.127,E2 -14007.127} C_VEL
LIN {X 0,Y 340.732,Z 143.665,A -85,B 0,C 180,E1 -14010.328,E2 -14010.328} C_VEL
LIN {X 0,Y 340.745,Z 143.663,A -85,B 0,C 180,E1 -14014.333,E2 -14014.333} C_VEL
LIN {X 0,Y 340.742,Z 143.668,A -85,B 0,C 180,E1 -14018.206,E2 -14018.206} C_VEL
LIN {X 0,Y 340.793,Z 143.655,A -85,B 0,C 180,E1 -14021.98,E2 -14021.98} C_VEL
LIN {X 0,Y 340.869,Z 143.646,A -85,B 0,C 180,E1 -14025.704,E2 -14025.704} C_VEL
LIN {X 0,Y 340.871,Z 143.649,A -85,B 0,C 180,E1 -14029.306,E2 -14029.306} C_VEL
LIN {X 0,Y 341.075,Z 143.624,A -85,B 0,C 180,E1 -14032.898,E2 -14032.898} C_VEL
LIN {X 0,Y 341.167,Z 143.606,A -85,B 0,C 180,E1 -14037.638,E2 -14037.638} C_VEL
LIN {X 0,Y 341.295,Z 143.597,A -85,B 0,C 180,E1 -14040,E2 -14040} C_VEL
LIN {X 0,Y 341.167,Z 143.608,A -85,B 0,C 180,E1 -14042.361,E2 -14042.361} C_VEL
LIN {X 0,Y 341.008,Z 143.635,A -85,B 0,C 180,E1 -14047.103,E2 -14047.103} C_VEL
LIN {X 0,Y 340.847,Z 143.653,A -85,B 0,C 180,E1 -14050.694,E2 -14050.694} C_VEL
LIN {X 0,Y 340.862,Z 143.65,A -85,B 0,C 180,E1 -14054.324,E2 -14054.324} C_VEL
LIN {X 0,Y 340.837,Z 143.654,A -85,B 0,C 180,E1 -14058.467,E2 -14058.467} C_VEL
LIN {X 0,Y 340.752,Z 143.663,A -85,B 0,C 180,E1 -14061.857,E2 -14061.857} C_VEL
LIN {X 0,Y 340.771,Z 143.658,A -85,B 0,C 180,E1 -14065.664,E2 -14065.664} C_VEL
LIN {X 0,Y 340.739,Z 143.666,A -85,B 0,C 180,E1 -14068.319,E2 -14068.319} C_VEL
LIN {X 0,Y 340.702,Z 143.67,A -85,B 0,C 180,E1 -14071.044,E2 -14071.044} C_VEL
LIN {X 0,Y 340.716,Z 143.666,A -85,B 0,C 180,E1 -14075.279,E2 -14075.279} C_VEL
LIN {X 0,Y 340.707,Z 143.65,A -85,B 0,C 180,E1 -14078.386,E2 -14078.386} C_VEL
LIN {X 0,Y 340.697,Z 143.662,A -85,B 0,C 180,E1 -14082.045,E2 -14082.045} C_VEL
LIN {X 0,Y 340.681,Z 143.672,A -85,B 0,C 180,E1 -14085.461,E2 -14085.461} C_VEL
LIN {X 0,Y 340.719,Z 143.79,A -85,B 0,C 180,E1 -14088.464,E2 -14088.464} C_VEL
LIN {X 0,Y 344.161,Z 154.455,A -85,B 0,C 180,E1 -14091.872,E2 -14091.872} C_VEL
LIN {X 0,Y 346.563,Z 162.795,A -85,B 0,C 180,E1 -14094.245,E2 -14094.245} C_VEL
LIN {X 0,Y 354.242,Z 177.013,A -85,B 0,C 180,E1 -14095.677,E2 -14095.677} C_VEL
LIN {X 0,Y 361.776,Z 192.529,A -85,B 0,C 180,E1 -14097.025,E2 -14097.025} C_VEL
LIN {X 0,Y 362.826,Z 196.555,A -85,B 0,C 180,E1 -14097.251,E2 -14097.251} C_VEL
LIN {X 0,Y 365.463,Z 211.198,A -85,B 0,C 180,E1 -14097.923,E2 -14097.923} C_VEL
LIN {X 0,Y 361.437,Z 330.062,A -85,B 0,C 180,E1 -14100.396,E2 -14100.396} C_VEL
LIN {X 0,Y 360.183,Z 345.687,A -85,B 0,C 180,E1 -14100.924,E2 -14100.924} C_VEL
LIN {X 0,Y 358.593,Z 360.111,A -85,B 0,C 180,E1 -14101.623,E2 -14101.623} C_VEL
LIN {X 0,Y 356.668,Z 374.552,A -85,B 0,C 180,E1 -14102.561,E2 -14102.561} C_VEL
LIN {X 0,Y 354.618,Z 387.962,A -85,B 0,C 180,E1 -14103.677,E2 -14103.677} C_VEL
LIN {X 0,Y 352.163,Z 401.523,A -85,B 0,C 180,E1 -14105.066,E2 -14105.066} C_VEL
LIN {X 0,Y 349.8,Z 413.839,A -85,B 0,C 180,E1 -14106.622,E2 -14106.622} C_VEL
LIN {X 0,Y 347.456,Z 425.104,A -85,B 0,C 180,E1 -14108.338,E2 -14108.338} C_VEL
LIN {X 0,Y 345.244,Z 436.103,A -85,B 0,C 180,E1 -14110.374,E2 -14110.374} C_VEL
LIN {X 0,Y 343.361,Z 445.248,A -85,B 0,C 180,E1 -14112.428,E2 -14112.428} C_VEL
LIN {X 0,Y 341.625,Z 453.994,A -85,B 0,C 180,E1 -14114.825,E2 -14114.825} C_VEL
LIN {X 0,Y 340.586,Z 460.051,A -85,B 0,C 180,E1 -14116.881,E2 -14116.881} C_VEL
LIN {X 0,Y 339.722,Z 465.742,A -85,B 0,C 180,E1 -14119.27,E2 -14119.27} C_VEL
LIN {X 0,Y 339.289,Z 470.111,A -85,B 0,C 180,E1 -14121.663,E2 -14121.663} C_VEL
LIN {X 0,Y 339.078,Z 473.398,A -85,B 0,C 180,E1 -14124.2,E2 -14124.2} C_VEL
LIN {X 0,Y 339.035,Z 475.207,A -85,B 0,C 180,E1 -14126.435,E2 -14126.435} C_VEL
LIN {X 0,Y 339.013,Z 475.962,A -85,B 0,C 180,E1 -14128.813,E2 -14128.813} C_VEL
LIN {X 0,Y 339.017,Z 475.578,A -85,B 0,C 180,E1 -14131.188,E2 -14131.188} C_VEL
LIN {X 0,Y 339.041,Z 474.04,A -85,B 0,C 180,E1 -14133.566,E2 -14133.566} C_VEL
LIN {X 0,Y 339.127,Z 471.311,A -85,B 0,C 180,E1 -14135.948,E2 -14135.948} C_VEL
LIN {X 0,Y 339.27,Z 467.309,A -85,B 0,C 180,E1 -14138.338,E2 -14138.338} C_VEL
LIN {X 0,Y 339.613,Z 461.911,A -85,B 0,C 180,E1 -14140.734,E2 -14140.734} C_VEL
LIN {X 0,Y 340.404,Z 455.017,A -85,B 0,C 180,E1 -14143.127,E2 -14143.127} C_VEL
LIN {X 0,Y 341.3,Z 447.557,A -85,B 0,C 180,E1 -14145.222,E2 -14145.222} C_VEL
LIN {X 0,Y 342.542,Z 438.592,A -85,B 0,C 180,E1 -14147.308,E2 -14147.308} C_VEL
LIN {X 0,Y 343.998,Z 429.452,A -85,B 0,C 180,E1 -14149.08,E2 -14149.08} C_VEL
LIN {X 0,Y 345.549,Z 418.335,A -85,B 0,C 180,E1 -14150.897,E2 -14150.897} C_VEL
LIN {X 0,Y 347.494,Z 405.638,A -85,B 0,C 180,E1 -14152.599,E2 -14152.599} C_VEL
LIN {X 0,Y 349.262,Z 392.474,A -85,B 0,C 180,E1 -14154.047,E2 -14154.047} C_VEL
LIN {X 0,Y 350.982,Z 379.711,A -85,B 0,C 180,E1 -14155.183,E2 -14155.183} C_VEL
LIN {X 0,Y 352.571,Z 365.015,A -85,B 0,C 180,E1 -14156.233,E2 -14156.233} C_VEL
LIN {X 0,Y 353.89,Z 350,A -85,B 0,C 180,E1 -14157.047,E2 -14157.047} C_VEL
LIN {X 0,Y 354.981,Z 334.204,A -85,B 0,C 180,E1 -14157.648,E2 -14157.648} C_VEL
LIN {X 0,Y 355.69,Z 314.645,A -85,B 0,C 180,E1 -14158.108,E2 -14158.108} C_VEL
LIN {X 0,Y 358.452,Z 209.381,A -85,B 0,C 180,E1 -14160.242,E2 -14160.242} C_VEL
LIN {X 0,Y 353.674,Z 182.915,A -85,B 0,C 180,E1 -14161.222,E2 -14161.222} C_VEL
LIN {X 0,Y 345.693,Z 163.534,A -85,B 0,C 180,E1 -14162.376,E2 -14162.376} C_VEL
LIN {X 0,Y 342.419,Z 150.213,A -85,B 0,C 180,E1 -14165.553,E2 -14165.553} C_VEL
LIN {X 0,Y 340.75,Z 143.67,A -85,B 0,C 180,E1 -14167.199,E2 -14167.199} C_VEL
LIN {X 0,Y 340.686,Z 143.673,A -85,B 0,C 180,E1 -14171.31,E2 -14171.31} C_VEL
LIN {X 0,Y 340.643,Z 143.681,A -85,B 0,C 180,E1 -14174.546,E2 -14174.546} C_VEL
LIN {X 0,Y 340.701,Z 143.674,A -85,B 0,C 180,E1 -14177.955,E2 -14177.955} C_VEL
LIN {X 0,Y 340.734,Z 143.661,A -85,B 0,C 180,E1 -14181.773,E2 -14181.773} C_VEL
LIN {X 0,Y 340.725,Z 143.669,A -85,B 0,C 180,E1 -14185.596,E2 -14185.596} C_VEL
LIN {X 0,Y 340.697,Z 143.672,A -85,B 0,C 180,E1 -14188.956,E2 -14188.956} C_VEL
LIN {X 0,Y 340.722,Z 143.645,A -85,B 0,C 180,E1 -14193.013,E2 -14193.013} C_VEL
LIN {X 0,Y 340.746,Z 143.663,A -85,B 0,C 180,E1 -14195.638,E2 -14195.638} C_VEL
LIN {X 0,Y 340.738,Z 143.663,A -85,B 0,C 180,E1 -14199.474,E2 -14199.474} C_VEL
LIN {X 0,Y 340.796,Z 143.655,A -85,B 0,C 180,E1 -14201.981,E2 -14201.981} C_VEL
LIN {X 0,Y 340.874,Z 143.648,A -85,B 0,C 180,E1 -14205.706,E2 -14205.706} C_VEL
LIN {X 0,Y 340.852,Z 143.65,A -85,B 0,C 180,E1 -14209.306,E2 -14209.306} C_VEL
LIN {X 0,Y 341.006,Z 143.629,A -85,B 0,C 180,E1 -14212.897,E2 -14212.897} C_VEL
LIN {X 0,Y 340.816,Z 143.654,A -85,B 0,C 180,E1 -14215.269,E2 -14215.269} C_VEL
LIN {X 0,Y 341.129,Z 143.603,A -85,B 0,C 180,E1 -14217.639,E2 -14217.639} C_VEL
LIN {X 0,Y 341.092,Z 143.604,A -85,B 0,C 180,E1 -14221.181,E2 -14221.181} C_VEL
LIN {X 0,Y 341.122,Z 143.61,A -85,B 0,C 180,E1 -14222.362,E2 -14222.362} C_VEL
LIN {X 0,Y 340.994,Z 143.624,A -85,B 0,C 180,E1 -14226.481,E2 -14226.481} C_VEL
LIN {X 0,Y 340.884,Z 143.615,A -85,B 0,C 180,E1 -14229.494,E2 -14229.494} C_VEL
LIN {X 0,Y 340.819,Z 143.649,A -85,B 0,C 180,E1 -14233.111,E2 -14233.111} C_VEL
LIN {X 0,Y 340.721,Z 143.66,A -85,B 0,C 180,E1 -14236.785,E2 -14236.785} C_VEL
LIN {X 0,Y 340.689,Z 143.671,A -85,B 0,C 180,E1 -14239.273,E2 -14239.273} C_VEL
LIN {X 0,Y 340.68,Z 143.668,A -85,B 0,C 180,E1 -14243.077,E2 -14243.077} C_VEL
LIN {X 0,Y 340.674,Z 143.671,A -85,B 0,C 180,E1 -14245.673,E2 -14245.673} C_VEL
LIN {X 0,Y 340.676,Z 143.653,A -85,B 0,C 180,E1 -14248.326,E2 -14248.326} C_VEL
LIN {X 0,Y 340.695,Z 143.652,A -85,B 0,C 180,E1 -14251.046,E2 -14251.046} C_VEL
LIN {X 0,Y 340.72,Z 143.663,A -85,B 0,C 180,E1 -14255.279,E2 -14255.279} C_VEL
LIN {X 0,Y 340.697,Z 143.644,A -85,B 0,C 180,E1 -14258.382,E2 -14258.382} C_VEL
LIN {X 0,Y 340.698,Z 143.669,A -85,B 0,C 180,E1 -14262.044,E2 -14262.044} C_VEL
LIN {X 0,Y 340.654,Z 143.655,A -85,B 0,C 180,E1 -14266.227,E2 -14266.227} C_VEL
LIN {X 0,Y 340.676,Z 143.674,A -85,B 0,C 180,E1 -14268.688,E2 -14268.688} C_VEL
LIN {X 0,Y 340.724,Z 143.656,A -85,B 0,C 180,E1 -14271.771,E2 -14271.771} C_VEL
LIN {X 0,Y 340.728,Z 143.666,A -85,B 0,C 180,E1 -14275.595,E2 -14275.595} C_VEL
LIN {X 0,Y 340.699,Z 143.673,A -85,B 0,C 180,E1 -14278.955,E2 -14278.955} C_VEL
LIN {X 0,Y 340.723,Z 143.671,A -85,B 0,C 180,E1 -14283.012,E2 -14283.012} C_VEL
LIN {X 0,Y 340.711,Z 143.671,A -85,B 0,C 180,E1 -14286.925,E2 -14286.925} C_VEL
LIN {X 0,Y 340.768,Z 143.659,A -85,B 0,C 180,E1 -14290.732,E2 -14290.732} C_VEL
LIN {X 0,Y 340.823,Z 143.658,A -85,B 0,C 180,E1 -14294.45,E2 -14294.45} C_VEL
LIN {X 0,Y 340.864,Z 143.741,A -85,B 0,C 180,E1 -14295.438,E2 -14295.438} C_VEL
LIN {X 0,Y 341.824,Z 147.37,A -85,B 0,C 180,E1 -14296.389,E2 -14296.389} C_VEL
LIN {X 0,Y 355.311,Z 177.942,A -85,B 0,C 180,E1 -14298.262,E2 -14298.262} C_VEL
LIN {X 0,Y 358.911,Z 187.442,A -85,B 0,C 180,E1 -14298.768,E2 -14298.768} C_VEL
LIN {X 0,Y 355.584,Z 311.868,A -85,B 0,C 180,E1 -14301.317,E2 -14301.317} C_VEL
LIN {X 0,Y 354.706,Z 327.377,A -85,B 0,C 180,E1 -14301.848,E2 -14301.848} C_VEL
LIN {X 0,Y 353.605,Z 342.007,A -85,B 0,C 180,E1 -14302.577,E2 -14302.577} C_VEL
LIN {X 0,Y 352.12,Z 356.816,A -85,B 0,C 180,E1 -14303.553,E2 -14303.553} C_VEL
LIN {X 0,Y 350.61,Z 370.168,A -85,B 0,C 180,E1 -14304.68,E2 -14304.68} C_VEL
LIN {X 0,Y 348.951,Z 382.55,A -85,B 0,C 180,E1 -14305.957,E2 -14305.957} C_VEL
LIN {X 0,Y 347.158,Z 395.128,A -85,B 0,C 180,E1 -14307.534,E2 -14307.534} C_VEL
LIN {X 0,Y 345.58,Z 405.671,A -85,B 0,C 180,E1 -14309.126,E2 -14309.126} C_VEL
LIN {X 0,Y 344.139,Z 415.421,A -85,B 0,C 180,E1 -14310.873,E2 -14310.873} C_VEL
LIN {X 0,Y 342.601,Z 425.06,A -85,B 0,C 180,E1 -14312.939,E2 -14312.939} C_VEL
LIN {X 0,Y 341.442,Z 433.062,A -85,B 0,C 180,E1 -14315.018,E2 -14315.018} C_VEL
LIN {X 0,Y 340.605,Z 439.717,A -85,B 0,C 180,E1 -14317.111,E2 -14317.111} C_VEL
LIN {X 0,Y 339.802,Z 445.857,A -85,B 0,C 180,E1 -14319.524,E2 -14319.524} C_VEL
LIN {X 0,Y 339.339,Z 450.569,A -85,B 0,C 180,E1 -14321.953,E2 -14321.953} C_VEL
LIN {X 0,Y 338.957,Z 453.968,A -85,B 0,C 180,E1 -14324.407,E2 -14324.407} C_VEL
LIN {X 0,Y 338.875,Z 456.104,A -85,B 0,C 180,E1 -14326.878,E2 -14326.878} C_VEL
LIN {X 0,Y 338.809,Z 457.011,A -85,B 0,C 180,E1 -14329.383,E2 -14329.383} C_VEL
LIN {X 0,Y 338.907,Z 456.657,A -85,B 0,C 180,E1 -14331.917,E2 -14331.917} C_VEL
LIN {X 0,Y 339.177,Z 454.997,A -85,B 0,C 180,E1 -14334.482,E2 -14334.482} C_VEL
LIN {X 0,Y 339.742,Z 451.789,A -85,B 0,C 180,E1 -14337.187,E2 -14337.187} C_VEL
LIN {X 0,Y 340.018,Z 449.76,A -85,B 0,C 180,E1 -14338.454,E2 -14338.454} C_VEL
LIN {X 0,Y 339.661,Z 448.099,A -85,B 0,C 180,E1 -14339.407,E2 -14339.407} C_VEL
LIN {X 0,Y 337.413,Z 445.186,A -85,B 0,C 180,E1 -14340.968,E2 -14340.968} C_VEL
LIN {X 0,Y 335.596,Z 442.549,A -85,B 0,C 180,E1 -14342.208,E2 -14342.208} C_VEL
LIN {X 0,Y 335.077,Z 440.275,A -85,B 0,C 180,E1 -14343.137,E2 -14343.137} C_VEL
LIN {X 0,Y 335.179,Z 439.403,A -85,B 0,C 180,E1 -14343.441,E2 -14343.441} C_VEL
LIN {X 0,Y 336.783,Z 432.148,A -85,B 0,C 180,E1 -14345.754,E2 -14345.754} C_VEL
LIN {X 0,Y 338.765,Z 423.565,A -85,B 0,C 180,E1 -14347.968,E2 -14347.968} C_VEL
LIN {X 0,Y 340.943,Z 413.664,A -85,B 0,C 180,E1 -14350.068,E2 -14350.068} C_VEL
LIN {X 0,Y 343.322,Z 403.147,A -85,B 0,C 180,E1 -14351.901,E2 -14351.901} C_VEL
LIN {X 0,Y 345.888,Z 390.65,A -85,B 0,C 180,E1 -14353.696,E2 -14353.696} C_VEL
LIN {X 0,Y 348.429,Z 377.387,A -85,B 0,C 180,E1 -14355.239,E2 -14355.239} C_VEL
LIN {X 0,Y 350.671,Z 363.67,A -85,B 0,C 180,E1 -14356.534,E2 -14356.534} C_VEL
LIN {X 0,Y 352.551,Z 350.514,A -85,B 0,C 180,E1 -14357.526,E2 -14357.526} C_VEL
LIN {X 0,Y 354.244,Z 335.231,A -85,B 0,C 180,E1 -14358.418,E2 -14358.418} C_VEL
LIN {X 0,Y 355.587,Z 320.019,A -85,B 0,C 180,E1 -14359.049,E2 -14359.049} C_VEL
LIN {X 0,Y 356.427,Z 303.385,A -85,B 0,C 180,E1 -14359.496,E2 -14359.496} C_VEL
LIN {X 0,Y 360.228,Z 194.64,A -85,B 0,C 180,E1 -14361.769,E2 -14361.769} C_VEL
LIN {X 0,Y 353.471,Z 180.457,A -85,B 0,C 180,E1 -14362.991,E2 -14362.991} C_VEL
LIN {X 0,Y 345.411,Z 165.785,A -85,B 0,C 180,E1 -14364.493,E2 -14364.493} C_VEL
LIN {X 0,Y 339.723,Z 156.544,A -85,B 0,C 180,E1 -14365.586,E2 -14365.586} C_VEL
LIN {X 0,Y 334.962,Z 148.685,A -85,B 0,C 180,E1 -14366.58,E2 -14366.58} C_VEL
LIN {X 0,Y 333.643,Z 144.537,A -85,B 0,C 180,E1 -14368.135,E2 -14368.135} C_VEL
LIN {X 0,Y 333.67,Z 144.534,A -85,B 0,C 180,E1 -14371.023,E2 -14371.023} C_VEL
LIN {X 0,Y 333.714,Z 144.527,A -85,B 0,C 180,E1 -14375.089,E2 -14375.089} C_VEL
LIN {X 0,Y 333.674,Z 144.544,A -85,B 0,C 180,E1 -14379.018,E2 -14379.018} C_VEL
LIN {X 0,Y 333.742,Z 144.536,A -85,B 0,C 180,E1 -14381.586,E2 -14381.586} C_VEL
LIN {X 0,Y 333.808,Z 144.525,A -85,B 0,C 180,E1 -14385.576,E2 -14385.576} C_VEL
LIN {X 0,Y 333.834,Z 144.524,A -85,B 0,C 180,E1 -14389.078,E2 -14389.078} C_VEL
LIN {X 0,Y 334.025,Z 144.502,A -85,B 0,C 180,E1 -14392.747,E2 -14392.747} C_VEL
LIN {X 0,Y 333.807,Z 144.522,A -85,B 0,C 180,E1 -14395.169,E2 -14395.169} C_VEL
LIN {X 0,Y 334.104,Z 144.486,A -85,B 0,C 180,E1 -14397.588,E2 -14397.588} C_VEL
LIN {X 0,Y 334.246,Z 144.475,A -85,B 0,C 180,E1 -14400,E2 -14400} C_VEL
LIN {X 0,Y 334.104,Z 144.488,A -85,B 0,C 180,E1 -14402.411,E2 -14402.411} C_VEL
LIN {X 0,Y 333.997,Z 144.502,A -85,B 0,C 180,E1 -14406.039,E2 -14406.039} C_VEL
LIN {X 0,Y 333.82,Z 144.524,A -85,B 0,C 180,E1 -14409.696,E2 -14409.696} C_VEL
LIN {X 0,Y 333.796,Z 144.527,A -85,B 0,C 180,E1 -14413.391,E2 -14413.391} C_VEL
LIN {X 0,Y 333.746,Z 144.534,A -85,B 0,C 180,E1 -14417.146,E2 -14417.146} C_VEL
LIN {X 0,Y 333.74,Z 144.529,A -85,B 0,C 180,E1 -14419.69,E2 -14419.69} C_VEL
LIN {X 0,Y 333.691,Z 144.541,A -85,B 0,C 180,E1 -14422.278,E2 -14422.278} C_VEL
LIN {X 0,Y 333.734,Z 144.532,A -85,B 0,C 180,E1 -14426.246,E2 -14426.246} C_VEL
LIN {X 0,Y 333.709,Z 144.536,A -85,B 0,C 180,E1 -14428.972,E2 -14428.972} C_VEL
LIN {X 0,Y 333.641,Z 144.546,A -85,B 0,C 180,E1 -14432.587,E2 -14432.587} C_VEL
LIN {X 0,Y 333.674,Z 144.547,A -85,B 0,C 180,E1 -14436.139,E2 -14436.139} C_VEL
LIN {X 0,Y 333.644,Z 144.531,A -85,B 0,C 180,E1 -14439.192,E2 -14439.192} C_VEL
LIN {X 0,Y 333.631,Z 144.537,A -85,B 0,C 180,E1 -14442.5,E2 -14442.5} C_VEL
LIN {X 0,Y 333.618,Z 144.544,A -85,B 0,C 180,E1 -14445.959,E2 -14445.959} C_VEL
LIN {X 0,Y 333.666,Z 144.725,A -85,B 0,C 180,E1 -14447.493,E2 -14447.493} C_VEL
LIN {X 0,Y 336.949,Z 154.95,A -85,B 0,C 180,E1 -14450.898,E2 -14450.898} C_VEL
LIN {X 0,Y 339.227,Z 162.412,A -85,B 0,C 180,E1 -14453.164,E2 -14453.164} C_VEL
LIN {X 0,Y 341.881,Z 167.067,A -85,B 0,C 180,E1 -14453.69,E2 -14453.69} C_VEL
LIN {X 0,Y 349.634,Z 181.523,A -85,B 0,C 180,E1 -14455.181,E2 -14455.181} C_VEL
LIN {X 0,Y 356.789,Z 196.41,A -85,B 0,C 180,E1 -14456.508,E2 -14456.508} C_VEL
LIN {X 0,Y 359.725,Z 212.51,A -85,B 0,C 180,E1 -14457.279,E2 -14457.279} C_VEL
LIN {X 0,Y 355.633,Z 329.107,A -85,B 0,C 180,E1 -14459.74,E2 -14459.74} C_VEL
LIN {X 0,Y 354.438,Z 344.159,A -85,B 0,C 180,E1 -14460.243,E2 -14460.243} C_VEL
LIN {X 0,Y 352.686,Z 358.911,A -85,B 0,C 180,E1 -14460.941,E2 -14460.941} C_VEL
LIN {X 0,Y 350.87,Z 372.73,A -85,B 0,C 180,E1 -14461.837,E2 -14461.837} C_VEL
LIN {X 0,Y 348.826,Z 385.573,A -85,B 0,C 180,E1 -14462.881,E2 -14462.881} C_VEL
LIN {X 0,Y 346.516,Z 398.251,A -85,B 0,C 180,E1 -14464.148,E2 -14464.148} C_VEL
LIN {X 0,Y 344.163,Z 410.032,A -85,B 0,C 180,E1 -14465.575,E2 -14465.575} C_VEL
LIN {X 0,Y 341.653,Z 421.88,A -85,B 0,C 180,E1 -14467.313,E2 -14467.313} C_VEL
LIN {X 0,Y 339.382,Z 432.327,A -85,B 0,C 180,E1 -14469.166,E2 -14469.166} C_VEL
LIN {X 0,Y 337.321,Z 441.695,A -85,B 0,C 180,E1 -14471.16,E2 -14471.16} C_VEL
LIN {X 0,Y 335.36,Z 450.937,A -85,B 0,C 180,E1 -14473.566,E2 -14473.566} C_VEL
LIN {X 0,Y 333.868,Z 458.45,A -85,B 0,C 180,E1 -14475.991,E2 -14475.991} C_VEL
LIN {X 0,Y 332.927,Z 464.458,A -85,B 0,C 180,E1 -14478.432,E2 -14478.432} C_VEL
LIN {X 0,Y 332.323,Z 469.106,A -85,B 0,C 180,E1 -14480.874,E2 -14480.874} C_VEL
LIN {X 0,Y 332.054,Z 471.728,A -85,B 0,C 180,E1 -14482.705,E2 -14482.705} C_VEL
LIN {X 0,Y 331.915,Z 474.234,A -85,B 0,C 180,E1 -14485.142,E2 -14485.142} C_VEL
LIN {X 0,Y 331.902,Z 475.556,A -85,B 0,C 180,E1 -14487.573,E2 -14487.573} C_VEL
LIN {X 0,Y 331.968,Z 475.705,A -85,B 0,C 180,E1 -14490,E2 -14490} C_VEL
LIN {X 0,Y 331.906,Z 474.705,A -85,B 0,C 180,E1 -14492.428,E2 -14492.428} C_VEL
LIN {X 0,Y 331.937,Z 472.536,A -85,B 0,C 180,E1 -14494.859,E2 -14494.859} C_VEL
LIN {X 0,Y 332.133,Z 469.144,A -85,B 0,C 180,E1 -14497.295,E2 -14497.295} C_VEL
LIN {X 0,Y 332.337,Z 464.419,A -85,B 0,C 180,E1 -14499.741,E2 -14499.741} C_VEL
LIN {X 0,Y 332.993,Z 458.246,A -85,B 0,C 180,E1 -14502.185,E2 -14502.185} C_VEL
LIN {X 0,Y 333.869,Z 450.452,A -85,B 0,C 180,E1 -14504.632,E2 -14504.632} C_VEL
LIN {X 0,Y 335.038,Z 442.105,A -85,B 0,C 180,E1 -14506.765,E2 -14506.765} C_VEL
LIN {X 0,Y 336.676,Z 432.069,A -85,B 0,C 180,E1 -14508.879,E2 -14508.879} C_VEL
LIN {X 0,Y 338.481,Z 420.051,A -85,B 0,C 180,E1 -14510.956,E2 -14510.956} C_VEL
LIN {X 0,Y 340.319,Z 408.337,A -85,B 0,C 180,E1 -14512.621,E2 -14512.621} C_VEL
LIN {X 0,Y 342.116,Z 395.788,A -85,B 0,C 180,E1 -14514.098,E2 -14514.098} C_VEL
LIN {X 0,Y 344.057,Z 382.067,A -85,B 0,C 180,E1 -14515.402,E2 -14515.402} C_VEL
LIN {X 0,Y 345.69,Z 367.946,A -85,B 0,C 180,E1 -14516.479,E2 -14516.479} C_VEL
LIN {X 0,Y 347.011,Z 353.832,A -85,B 0,C 180,E1 -14517.314,E2 -14517.314} C_VEL
LIN {X 0,Y 348.304,Z 338.193,A -85,B 0,C 180,E1 -14517.979,E2 -14517.979} C_VEL
LIN {X 0,Y 348.992,Z 322.819,A -85,B 0,C 180,E1 -14518.409,E2 -14518.409} C_VEL
LIN {X 0,Y 352.068,Z 210.425,A -85,B 0,C 180,E1 -14520.727,E2 -14520.727} C_VEL
LIN {X 0,Y 347.774,Z 185.873,A -85,B 0,C 180,E1 -14521.649,E2 -14521.649} C_VEL
LIN {X 0,Y 338.435,Z 163.339,A -85,B 0,C 180,E1 -14523.026,E2 -14523.026} C_VEL
LIN {X 0,Y 334.801,Z 148.807,A -85,B 0,C 180,E1 -14526.605,E2 -14526.605} C_VEL
LIN {X 0,Y 333.691,Z 144.544,A -85,B 0,C 180,E1 -14527.742,E2 -14527.742} C_VEL
LIN {X 0,Y 333.647,Z 144.55,A -85,B 0,C 180,E1 -14530.768,E2 -14530.768} C_VEL
LIN {X 0,Y 333.595,Z 144.559,A -85,B 0,C 180,E1 -14534.251,E2 -14534.251} C_VEL
LIN {X 0,Y 333.643,Z 144.553,A -85,B 0,C 180,E1 -14537.619,E2 -14537.619} C_VEL
LIN {X 0,Y 333.654,Z 144.539,A -85,B 0,C 180,E1 -14541.203,E2 -14541.203} C_VEL
LIN {X 0,Y 333.678,Z 144.543,A -85,B 0,C 180,E1 -14543.862,E2 -14543.862} C_VEL
LIN {X 0,Y 333.646,Z 144.547,A -85,B 0,C 180,E1 -14547.414,E2 -14547.414} C_VEL
LIN {X 0,Y 333.657,Z 144.532,A -85,B 0,C 180,E1 -14551.023,E2 -14551.023} C_VEL
LIN {X 0,Y 333.699,Z 144.538,A -85,B 0,C 180,E1 -14555.089,E2 -14555.089} C_VEL
LIN {X 0,Y 333.677,Z 144.541,A -85,B 0,C 180,E1 -14559.019,E2 -14559.019} C_VEL
LIN {X 0,Y 333.745,Z 144.533,A -85,B 0,C 180,E1 -14561.587,E2 -14561.587} C_VEL
LIN {X 0,Y 333.812,Z 144.527,A -85,B 0,C 180,E1 -14565.577,E2 -14565.577} C_VEL
LIN {X 0,Y 333.822,Z 144.527,A -85,B 0,C 180,E1 -14569.078,E2 -14569.078} C_VEL
LIN {X 0,Y 333.961,Z 144.506,A -85,B 0,C 180,E1 -14572.747,E2 -14572.747} C_VEL
LIN {X 0,Y 333.783,Z 144.53,A -85,B 0,C 180,E1 -14575.169,E2 -14575.169} C_VEL
LIN {X 0,Y 334.07,Z 144.483,A -85,B 0,C 180,E1 -14577.589,E2 -14577.589} C_VEL
LIN {X 0,Y 334.062,Z 144.479,A -85,B 0,C 180,E1 -14581.206,E2 -14581.206} C_VEL
LIN {X 0,Y 334.062,Z 144.489,A -85,B 0,C 180,E1 -14582.412,E2 -14582.412} C_VEL
LIN {X 0,Y 333.963,Z 144.5,A -85,B 0,C 180,E1 -14586.473,E2 -14586.473} C_VEL
LIN {X 0,Y 333.821,Z 144.494,A -85,B 0,C 180,E1 -14589.697,E2 -14589.697} C_VEL
LIN {X 0,Y 333.765,Z 144.53,A -85,B 0,C 180,E1 -14593.393,E2 -14593.393} C_VEL
LIN {X 0,Y 333.67,Z 144.538,A -85,B 0,C 180,E1 -14597.151,E2 -14597.151} C_VEL
LIN {X 0,Y 333.631,Z 144.553,A -85,B 0,C 180,E1 -14599.697,E2 -14599.697} C_VEL
LIN {X 0,Y 333.625,Z 144.544,A -85,B 0,C 180,E1 -14602.284,E2 -14602.284} C_VEL
LIN {X 0,Y 333.662,Z 144.548,A -85,B 0,C 180,E1 -14605.078,E2 -14605.078} C_VEL
LIN {X 0,Y 333.628,Z 144.523,A -85,B 0,C 180,E1 -14608.981,E2 -14608.981} C_VEL
LIN {X 0,Y 333.648,Z 144.543,A -85,B 0,C 180,E1 -14612.587,E2 -14612.587} C_VEL
LIN {X 0,Y 333.678,Z 144.537,A -85,B 0,C 180,E1 -14616.139,E2 -14616.139} C_VEL
LIN {X 0,Y 333.606,Z 144.533,A -85,B 0,C 180,E1 -14619.199,E2 -14619.199} C_VEL
LIN {X 0,Y 333.633,Z 144.551,A -85,B 0,C 180,E1 -14622.499,E2 -14622.499} C_VEL
LIN {X 0,Y 333.598,Z 144.533,A -85,B 0,C 180,E1 -14625.954,E2 -14625.954} C_VEL
LIN {X 0,Y 333.607,Z 144.554,A -85,B 0,C 180,E1 -14629.324,E2 -14629.324} C_VEL
LIN {X 0,Y 333.668,Z 144.538,A -85,B 0,C 180,E1 -14633.168,E2 -14633.168} C_VEL
LIN {X 0,Y 333.679,Z 144.544,A -85,B 0,C 180,E1 -14635.341,E2 -14635.341} C_VEL
LIN {X 0,Y 333.634,Z 144.543,A -85,B 0,C 180,E1 -14638.222,E2 -14638.222} C_VEL
LIN {X 0,Y 333.659,Z 144.544,A -85,B 0,C 180,E1 -14641.022,E2 -14641.022} C_VEL
LIN {X 0,Y 333.671,Z 144.549,A -85,B 0,C 180,E1 -14645.086,E2 -14645.086} C_VEL
LIN {X 0,Y 333.671,Z 144.546,A -85,B 0,C 180,E1 -14649.018,E2 -14649.018} C_VEL
LIN {X 0,Y 333.747,Z 144.52,A -85,B 0,C 180,E1 -14651.586,E2 -14651.586} C_VEL
LIN {X 0,Y 333.797,Z 144.566,A -85,B 0,C 180,E1 -14654.913,E2 -14654.913} C_VEL
LIN {X 0,Y 334.645,Z 147.748,A -85,B 0,C 180,E1 -14655.731,E2 -14655.731} C_VEL
LIN {X 0,Y 346.029,Z 173.027,A -85,B 0,C 180,E1 -14657.369,E2 -14657.369} C_VEL
LIN {X 0,Y 352.493,Z 188.919,A -85,B 0,C 180,E1 -14658.28,E2 -14658.28} C_VEL
LIN {X 0,Y 349.113,Z 311.77,A -85,B 0,C 180,E1 -14660.841,E2 -14660.841} C_VEL
LIN {X 0,Y 348.239,Z 327.006,A -85,B 0,C 180,E1 -14661.366,E2 -14661.366} C_VEL
LIN {X 0,Y 347.147,Z 341.155,A -85,B 0,C 180,E1 -14662.072,E2 -14662.072} C_VEL
LIN {X 0,Y 345.753,Z 355.203,A -85,B 0,C 180,E1 -14662.994,E2 -14662.994} C_VEL
LIN {X 0,Y 344.154,Z 368.927,A -85,B 0,C 180,E1 -14664.139,E2 -14664.139} C_VEL
LIN {X 0,Y 342.451,Z 381.562,A -85,B 0,C 180,E1 -14665.438,E2 -14665.438} C_VEL
LIN {X 0,Y 340.54,Z 394.357,A -85,B 0,C 180,E1 -14667.042,E2 -14667.042} C_VEL
LIN {X 0,Y 338.735,Z 405.954,A -85,B 0,C 180,E1 -14668.811,E2 -14668.811} C_VEL
LIN {X 0,Y 337.038,Z 416.881,A -85,B 0,C 180,E1 -14670.831,E2 -14670.831} C_VEL
LIN {X 0,Y 335.467,Z 426.552,A -85,B 0,C 180,E1 -14673.002,E2 -14673.002} C_VEL
LIN {X 0,Y 334.297,Z 434.327,A -85,B 0,C 180,E1 -14675.126,E2 -14675.126} C_VEL
LIN {X 0,Y 333.446,Z 440.78,A -85,B 0,C 180,E1 -14677.265,E2 -14677.265} C_VEL
LIN {X 0,Y 332.672,Z 446.726,A -85,B 0,C 180,E1 -14679.73,E2 -14679.73} C_VEL
LIN {X 0,Y 332.184,Z 451.273,A -85,B 0,C 180,E1 -14682.214,E2 -14682.214} C_VEL
LIN {X 0,Y 331.835,Z 454.529,A -85,B 0,C 180,E1 -14684.723,E2 -14684.723} C_VEL
LIN {X 0,Y 331.774,Z 456.525,A -85,B 0,C 180,E1 -14687.251,E2 -14687.251} C_VEL
LIN {X 0,Y 331.72,Z 457.261,A -85,B 0,C 180,E1 -14689.815,E2 -14689.815} C_VEL
LIN {X 0,Y 331.845,Z 456.728,A -85,B 0,C 180,E1 -14692.408,E2 -14692.408} C_VEL
LIN {X 0,Y 332.168,Z 454.885,A -85,B 0,C 180,E1 -14695.034,E2 -14695.034} C_VEL
LIN {X 0,Y 332.765,Z 451.648,A -85,B 0,C 180,E1 -14697.687,E2 -14697.687} C_VEL
LIN {X 0,Y 333.617,Z 446.897,A -85,B 0,C 180,E1 -14700.37,E2 -14700.37} C_VEL
LIN {X 0,Y 334.953,Z 440.486,A -85,B 0,C 180,E1 -14703.061,E2 -14703.061} C_VEL
LIN {X 0,Y 335.179,Z 439.403,A -85,B 0,C 180,E1 -14703.441,E2 -14703.441} C_VEL
LIN {X 0,Y 335.111,Z 436.885,A -85,B 0,C 180,E1 -14704.351,E2 -14704.351} C_VEL
LIN {X 0,Y 331.95,Z 429.007,A -85,B 0,C 180,E1 -14707.05,E2 -14707.05} C_VEL
LIN {X 0,Y 331.708,Z 425.9,A -85,B 0,C 180,E1 -14707.923,E2 -14707.923} C_VEL
LIN {X 0,Y 331.895,Z 424.801,A -85,B 0,C 180,E1 -14708.206,E2 -14708.206} C_VEL
LIN {X 0,Y 334.13,Z 415.327,A -85,B 0,C 180,E1 -14710.299,E2 -14710.299} C_VEL
LIN {X 0,Y 336.729,Z 404.259,A -85,B 0,C 180,E1 -14712.306,E2 -14712.306} C_VEL
LIN {X 0,Y 339.318,Z 392.349,A -85,B 0,C 180,E1 -14714.08,E2 -14714.08} C_VEL
LIN {X 0,Y 341.999,Z 379.185,A -85,B 0,C 180,E1 -14715.677,E2 -14715.677} C_VEL
LIN {X 0,Y 344.471,Z 365.179,A -85,B 0,C 180,E1 -14717.048,E2 -14717.048} C_VEL
LIN {X 0,Y 346.447,Z 351.921,A -85,B 0,C 180,E1 -14718.08,E2 -14718.08} C_VEL
LIN {X 0,Y 348.188,Z 337.303,A -85,B 0,C 180,E1 -14718.972,E2 -14718.972} C_VEL
LIN {X 0,Y 349.63,Z 322.187,A -85,B 0,C 180,E1 -14719.637,E2 -14719.637} C_VEL
LIN {X 0,Y 350.557,Z 306.583,A -85,B 0,C 180,E1 -14720.093,E2 -14720.093} C_VEL
LIN {X 0,Y 354.557,Z 196.967,A -85,B 0,C 180,E1 -14722.418,E2 -14722.418} C_VEL
LIN {X 0,Y 347.66,Z 182.52,A -85,B 0,C 180,E1 -14723.719,E2 -14723.719} C_VEL
LIN {X 0,Y 338.491,Z 166.183,A -85,B 0,C 180,E1 -14725.497,E2 -14725.497} C_VEL
LIN {X 0,Y 330.217,Z 153.007,A -85,B 0,C 180,E1 -14727.212,E2 -14727.212} C_VEL
LIN {X 0,Y 327.652,Z 148.953,A -85,B 0,C 180,E1 -14727.799,E2 -14727.799} C_VEL
LIN {X 0,Y 326.6,Z 145.42,A -85,B 0,C 180,E1 -14729.133,E2 -14729.133} C_VEL
LIN {X 0,Y 326.628,Z 145.419,A -85,B 0,C 180,E1 -14733.137,E2 -14733.137} C_VEL
LIN {X 0,Y 326.644,Z 145.401,A -85,B 0,C 180,E1 -14735.87,E2 -14735.87} C_VEL
LIN {X 0,Y 326.651,Z 145.417,A -85,B 0,C 180,E1 -14739.864,E2 -14739.864} C_VEL
LIN {X 0,Y 326.664,Z 145.415,A -85,B 0,C 180,E1 -14742.47,E2 -14742.47} C_VEL
LIN {X 0,Y 326.759,Z 145.409,A -85,B 0,C 180,E1 -14746.314,E2 -14746.314} C_VEL
LIN {X 0,Y 326.814,Z 145.399,A -85,B 0,C 180,E1 -14750.093,E2 -14750.093} C_VEL
LIN {X 0,Y 326.979,Z 145.38,A -85,B 0,C 180,E1 -14752.59,E2 -14752.59} C_VEL
LIN {X 0,Y 326.775,Z 145.398,A -85,B 0,C 180,E1 -14755.064,E2 -14755.064} C_VEL
LIN {X 0,Y 327.045,Z 145.365,A -85,B 0,C 180,E1 -14757.536,E2 -14757.536} C_VEL
LIN {X 0,Y 327.197,Z 145.353,A -85,B 0,C 180,E1 -14759.999,E2 -14759.999} C_VEL
LIN {X 0,Y 327.045,Z 145.368,A -85,B 0,C 180,E1 -14762.463,E2 -14762.463} C_VEL
LIN {X 0,Y 326.95,Z 145.381,A -85,B 0,C 180,E1 -14766.169,E2 -14766.169} C_VEL
LIN {X 0,Y 326.782,Z 145.402,A -85,B 0,C 180,E1 -14769.907,E2 -14769.907} C_VEL
LIN {X 0,Y 326.758,Z 145.406,A -85,B 0,C 180,E1 -14773.685,E2 -14773.685} C_VEL
LIN {X 0,Y 326.699,Z 145.416,A -85,B 0,C 180,E1 -14777.527,E2 -14777.527} C_VEL
LIN {X 0,Y 326.667,Z 145.411,A -85,B 0,C 180,E1 -14780.134,E2 -14780.134} C_VEL
LIN {X 0,Y 326.651,Z 145.419,A -85,B 0,C 180,E1 -14784.128,E2 -14784.128} C_VEL
LIN {X 0,Y 326.683,Z 145.412,A -85,B 0,C 180,E1 -14786.857,E2 -14786.857} C_VEL
LIN {X 0,Y 326.637,Z 145.424,A -85,B 0,C 180,E1 -14790.611,E2 -14790.611} C_VEL
LIN {X 0,Y 326.605,Z 145.428,A -85,B 0,C 180,E1 -14794.019,E2 -14794.019} C_VEL
LIN {X 0,Y 326.625,Z 145.416,A -85,B 0,C 180,E1 -14797.238,E2 -14797.238} C_VEL
LIN {X 0,Y 326.576,Z 145.433,A -85,B 0,C 180,E1 -14801.131,E2 -14801.131} C_VEL
LIN {X 0,Y 326.554,Z 145.432,A -85,B 0,C 180,E1 -14804.748,E2 -14804.748} C_VEL
LIN {X 0,Y 326.574,Z 145.419,A -85,B 0,C 180,E1 -14806.377,E2 -14806.377} C_VEL
LIN {X 0,Y 330.015,Z 155.972,A -85,B 0,C 180,E1 -14810.054,E2 -14810.054} C_VEL
LIN {X 0,Y 331.967,Z 162.196,A -85,B 0,C 180,E1 -14812.012,E2 -14812.012} C_VEL
LIN {X 0,Y 340.546,Z 177.343,A -85,B 0,C 180,E1 -14813.784,E2 -14813.784} C_VEL
LIN {X 0,Y 348.765,Z 193.546,A -85,B 0,C 180,E1 -14815.386,E2 -14815.386} C_VEL
LIN {X 0,Y 351.691,Z 199.956,A -85,B 0,C 180,E1 -14815.947,E2 -14815.947} C_VEL
LIN {X 0,Y 354.004,Z 213.568,A -85,B 0,C 180,E1 -14816.599,E2 -14816.599} C_VEL
LIN {X 0,Y 349.904,Z 326.912,A -85,B 0,C 180,E1 -14819.024,E2 -14819.024} C_VEL
LIN {X 0,Y 348.773,Z 341.792,A -85,B 0,C 180,E1 -14819.5,E2 -14819.5} C_VEL
LIN {X 0,Y 347.074,Z 356.492,A -85,B 0,C 180,E1 -14820.174,E2 -14820.174} C_VEL
LIN {X 0,Y 345.092,Z 371.244,A -85,B 0,C 180,E1 -14821.109,E2 -14821.109} C_VEL
LIN {X 0,Y 342.833,Z 384.763,A -85,B 0,C 180,E1 -14822.201,E2 -14822.201} C_VEL
LIN {X 0,Y 340.166,Z 398.816,A -85,B 0,C 180,E1 -14823.628,E2 -14823.628} C_VEL
LIN {X 0,Y 337.73,Z 410.467,A -85,B 0,C 180,E1 -14825.078,E2 -14825.078} C_VEL
LIN {X 0,Y 335.105,Z 422.21,A -85,B 0,C 180,E1 -14826.845,E2 -14826.845} C_VEL
LIN {X 0,Y 332.85,Z 432.003,A -85,B 0,C 180,E1 -14828.613,E2 -14828.613} C_VEL
LIN {X 0,Y 330.57,Z 441.862,A -85,B 0,C 180,E1 -14830.76,E2 -14830.76} C_VEL
LIN {X 0,Y 328.766,Z 450.014,A -85,B 0,C 180,E1 -14832.907,E2 -14832.907} C_VEL
LIN {X 0,Y 327.132,Z 457.118,A -85,B 0,C 180,E1 -14835.186,E2 -14835.186} C_VEL
LIN {X 0,Y 326.177,Z 463.055,A -85,B 0,C 180,E1 -14837.558,E2 -14837.558} C_VEL
LIN {X 0,Y 325.384,Z 467.973,A -85,B 0,C 180,E1 -14840.05,E2 -14840.05} C_VEL
LIN {X 0,Y 324.975,Z 471.626,A -85,B 0,C 180,E1 -14842.545,E2 -14842.545} C_VEL
LIN {X 0,Y 324.833,Z 474.088,A -85,B 0,C 180,E1 -14845.036,E2 -14845.036} C_VEL
LIN {X 0,Y 324.821,Z 475.388,A -85,B 0,C 180,E1 -14847.52,E2 -14847.52} C_VEL
LIN {X 0,Y 324.872,Z 475.494,A -85,B 0,C 180,E1 -14850,E2 -14850} C_VEL
LIN {X 0,Y 324.826,Z 474.45,A -85,B 0,C 180,E1 -14852.481,E2 -14852.481} C_VEL
LIN {X 0,Y 324.851,Z 472.235,A -85,B 0,C 180,E1 -14854.965,E2 -14854.965} C_VEL
LIN {X 0,Y 325.032,Z 468.793,A -85,B 0,C 180,E1 -14857.455,E2 -14857.455} C_VEL
LIN {X 0,Y 325.294,Z 464.022,A -85,B 0,C 180,E1 -14859.954,E2 -14859.954} C_VEL
LIN {X 0,Y 325.973,Z 457.799,A -85,B 0,C 180,E1 -14862.451,E2 -14862.451} C_VEL
LIN {X 0,Y 326.925,Z 449.935,A -85,B 0,C 180,E1 -14864.95,E2 -14864.95} C_VEL
LIN {X 0,Y 328.164,Z 441.543,A -85,B 0,C 180,E1 -14867.126,E2 -14867.126} C_VEL
LIN {X 0,Y 329.862,Z 431.423,A -85,B 0,C 180,E1 -14869.284,E2 -14869.284} C_VEL
LIN {X 0,Y 331.51,Z 421.033,A -85,B 0,C 180,E1 -14871.125,E2 -14871.125} C_VEL
LIN {X 0,Y 333.506,Z 408.639,A -85,B 0,C 180,E1 -14872.946,E2 -14872.946} C_VEL
LIN {X 0,Y 335.344,Z 396.17,A -85,B 0,C 180,E1 -14874.451,E2 -14874.451} C_VEL
LIN {X 0,Y 337.347,Z 382.583,A -85,B 0,C 180,E1 -14875.779,E2 -14875.779} C_VEL
LIN {X 0,Y 339.144,Z 367.716,A -85,B 0,C 180,E1 -14876.938,E2 -14876.938} C_VEL
LIN {X 0,Y 340.59,Z 352.745,A -85,B 0,C 180,E1 -14877.831,E2 -14877.831} C_VEL
LIN {X 0,Y 341.845,Z 337.677,A -85,B 0,C 180,E1 -14878.472,E2 -14878.472} C_VEL
LIN {X 0,Y 342.564,Z 322.082,A -85,B 0,C 180,E1 -14878.909,E2 -14878.909} C_VEL
LIN {X 0,Y 345.696,Z 211.416,A -85,B 0,C 180,E1 -14881.227,E2 -14881.227} C_VEL
LIN {X 0,Y 341.637,Z 188.245,A -85,B 0,C 180,E1 -14882.119,E2 -14882.119} C_VEL
LIN {X 0,Y 332.093,Z 165.624,A -85,B 0,C 180,E1 -14883.534,E2 -14883.534} C_VEL
LIN {X 0,Y 331.142,Z 163.231,A -85,B 0,C 180,E1 -14883.686,E2 -14883.686} C_VEL
LIN {X 0,Y 327.698,Z 149.433,A -85,B 0,C 180,E1 -14887.183,E2 -14887.183} C_VEL
LIN {X 0,Y 326.635,Z 145.421,A -85,B 0,C 180,E1 -14888.267,E2 -14888.267} C_VEL
LIN {X 0,Y 326.577,Z 145.434,A -85,B 0,C 180,E1 -14891.846,E2 -14891.846} C_VEL
LIN {X 0,Y 326.529,Z 145.442,A -85,B 0,C 180,E1 -14895.258,E2 -14895.258} C_VEL
LIN {X 0,Y 326.58,Z 145.433,A -85,B 0,C 180,E1 -14898.869,E2 -14898.869} C_VEL
LIN {X 0,Y 326.629,Z 145.422,A -85,B 0,C 180,E1 -14902.762,E2 -14902.762} C_VEL
LIN {X 0,Y 326.609,Z 145.425,A -85,B 0,C 180,E1 -14905.981,E2 -14905.981} C_VEL
LIN {X 0,Y 326.614,Z 145.424,A -85,B 0,C 180,E1 -14909.398,E2 -14909.398} C_VEL
LIN {X 0,Y 326.616,Z 145.402,A -85,B 0,C 180,E1 -14913.137,E2 -14913.137} C_VEL
LIN {X 0,Y 326.637,Z 145.42,A -85,B 0,C 180,E1 -14915.87,E2 -14915.87} C_VEL
LIN {X 0,Y 326.637,Z 145.419,A -85,B 0,C 180,E1 -14919.864,E2 -14919.864} C_VEL
LIN {X 0,Y 326.668,Z 145.413,A -85,B 0,C 180,E1 -14922.471,E2 -14922.471} C_VEL
LIN {X 0,Y 326.763,Z 145.408,A -85,B 0,C 180,E1 -14926.315,E2 -14926.315} C_VEL
LIN {X 0,Y 326.787,Z 145.404,A -85,B 0,C 180,E1 -14930.093,E2 -14930.093} C_VEL
LIN {X 0,Y 326.947,Z 145.381,A -85,B 0,C 180,E1 -14933.83,E2 -14933.83} C_VEL
LIN {X 0,Y 327.013,Z 145.362,A -85,B 0,C 180,E1 -14937.537,E2 -14937.537} C_VEL
LIN {X 0,Y 327.032,Z 145.355,A -85,B 0,C 180,E1 -14941.232,E2 -14941.232} C_VEL
LIN {X 0,Y 326.742,Z 145.406,A -85,B 0,C 180,E1 -14943.7,E2 -14943.7} C_VEL
LIN {X 0,Y 326.925,Z 145.375,A -85,B 0,C 180,E1 -14946.461,E2 -14946.461} C_VEL
LIN {X 0,Y 326.784,Z 145.371,A -85,B 0,C 180,E1 -14949.908,E2 -14949.908} C_VEL
LIN {X 0,Y 326.726,Z 145.409,A -85,B 0,C 180,E1 -14953.687,E2 -14953.687} C_VEL
LIN {X 0,Y 326.62,Z 145.418,A -85,B 0,C 180,E1 -14957.533,E2 -14957.533} C_VEL
LIN {X 0,Y 326.587,Z 145.427,A -85,B 0,C 180,E1 -14960.14,E2 -14960.14} C_VEL
LIN {X 0,Y 326.578,Z 145.422,A -85,B 0,C 180,E1 -14962.791,E2 -14962.791} C_VEL
LIN {X 0,Y 326.605,Z 145.425,A -85,B 0,C 180,E1 -14965.492,E2 -14965.492} C_VEL
LIN {X 0,Y 326.592,Z 145.406,A -85,B 0,C 180,E1 -14968.257,E2 -14968.257} C_VEL
LIN {X 0,Y 326.576,Z 145.41,A -85,B 0,C 180,E1 -14971.098,E2 -14971.098} C_VEL
LIN {X 0,Y 326.611,Z 145.423,A -85,B 0,C 180,E1 -14974.02,E2 -14974.02} C_VEL
LIN {X 0,Y 326.626,Z 145.4,A -85,B 0,C 180,E1 -14977.237,E2 -14977.237} C_VEL
LIN {X 0,Y 326.549,Z 145.431,A -85,B 0,C 180,E1 -14981.125,E2 -14981.125} C_VEL
LIN {X 0,Y 326.564,Z 145.426,A -85,B 0,C 180,E1 -14983.526,E2 -14983.526} C_VEL
LIN {X 0,Y 326.578,Z 145.416,A -85,B 0,C 180,E1 -14987.029,E2 -14987.029} C_VEL
LIN {X 0,Y 326.576,Z 145.423,A -85,B 0,C 180,E1 -14990.781,E2 -14990.781} C_VEL
LIN {X 0,Y 326.617,Z 145.425,A -85,B 0,C 180,E1 -14994.48,E2 -14994.48} C_VEL
LIN {X 0,Y 326.613,Z 145.413,A -85,B 0,C 180,E1 -14997.455,E2 -14997.455} C_VEL
LIN {X 0,Y 326.622,Z 145.426,A -85,B 0,C 180,E1 -15000.336,E2 -15000.336} C_VEL
LIN {X 0,Y 326.607,Z 145.43,A -85,B 0,C 180,E1 -15004.509,E2 -15004.509} C_VEL
LIN {X 0,Y 326.621,Z 145.426,A -85,B 0,C 180,E1 -15008.543,E2 -15008.543} C_VEL
LIN {X 0,Y 326.712,Z 145.401,A -85,B 0,C 180,E1 -15011.175,E2 -15011.175} C_VEL
LIN {X 0,Y 326.746,Z 145.512,A -85,B 0,C 180,E1 -15014.403,E2 -15014.403} C_VEL
LIN {X 0,Y 327.376,Z 147.897,A -85,B 0,C 180,E1 -15015.029,E2 -15015.029} C_VEL
LIN {X 0,Y 337.08,Z 168.912,A -85,B 0,C 180,E1 -15016.475,E2 -15016.475} C_VEL
LIN {X 0,Y 345.715,Z 189.572,A -85,B 0,C 180,E1 -15017.731,E2 -15017.731} C_VEL
LIN {X 0,Y 346.116,Z 191.326,A -85,B 0,C 180,E1 -15017.806,E2 -15017.806} C_VEL
LIN {X 0,Y 342.602,Z 312.793,A -85,B 0,C 180,E1 -15020.382,E2 -15020.382} C_VEL
LIN {X 0,Y 341.683,Z 328.37,A -85,B 0,C 180,E1 -15020.944,E2 -15020.944} C_VEL
LIN {X 0,Y 340.498,Z 342.801,A -85,B 0,C 180,E1 -15021.692,E2 -15021.692} C_VEL
LIN {X 0,Y 338.913,Z 357.525,A -85,B 0,C 180,E1 -15022.702,E2 -15022.702} C_VEL
LIN {X 0,Y 337.326,Z 370.826,A -85,B 0,C 180,E1 -15023.87,E2 -15023.87} C_VEL
LIN {X 0,Y 335.367,Z 384.455,A -85,B 0,C 180,E1 -15025.342,E2 -15025.342} C_VEL
LIN {X 0,Y 333.433,Z 396.79,A -85,B 0,C 180,E1 -15026.979,E2 -15026.979} C_VEL
LIN {X 0,Y 331.625,Z 408.017,A -85,B 0,C 180,E1 -15028.785,E2 -15028.785} C_VEL
LIN {X 0,Y 329.948,Z 418.33,A -85,B 0,C 180,E1 -15030.785,E2 -15030.785} C_VEL
LIN {X 0,Y 328.305,Z 428.048,A -85,B 0,C 180,E1 -15033.067,E2 -15033.067} C_VEL
LIN {X 0,Y 327.153,Z 435.59,A -85,B 0,C 180,E1 -15035.238,E2 -15035.238} C_VEL
LIN {X 0,Y 326.186,Z 442.396,A -85,B 0,C 180,E1 -15037.638,E2 -15037.638} C_VEL
LIN {X 0,Y 325.524,Z 447.589,A -85,B 0,C 180,E1 -15039.945,E2 -15039.945} C_VEL
LIN {X 0,Y 325.053,Z 451.954,A -85,B 0,C 180,E1 -15042.486,E2 -15042.486} C_VEL
LIN {X 0,Y 324.708,Z 455.037,A -85,B 0,C 180,E1 -15045.054,E2 -15045.054} C_VEL
LIN {X 0,Y 324.668,Z 456.907,A -85,B 0,C 180,E1 -15047.736,E2 -15047.736} C_VEL
LIN {X 0,Y 324.634,Z 457.468,A -85,B 0,C 180,E1 -15050.266,E2 -15050.266} C_VEL
LIN {X 0,Y 324.806,Z 456.788,A -85,B 0,C 180,E1 -15052.921,E2 -15052.921} C_VEL
LIN {X 0,Y 325.179,Z 454.771,A -85,B 0,C 180,E1 -15055.61,E2 -15055.61} C_VEL
LIN {X 0,Y 325.844,Z 451.339,A -85,B 0,C 180,E1 -15058.327,E2 -15058.327} C_VEL
LIN {X 0,Y 326.833,Z 446.377,A -85,B 0,C 180,E1 -15061.069,E2 -15061.069} C_VEL
LIN {X 0,Y 328.228,Z 440.175,A -85,B 0,C 180,E1 -15063.64,E2 -15063.64} C_VEL
LIN {X 0,Y 329.839,Z 433.259,A -85,B 0,C 180,E1 -15065.934,E2 -15065.934} C_VEL
LIN {X 0,Y 331.895,Z 424.801,A -85,B 0,C 180,E1 -15068.206,E2 -15068.206} C_VEL
LIN {X 0,Y 332.07,Z 421.507,A -85,B 0,C 180,E1 -15069.054,E2 -15069.054} C_VEL
LIN {X 0,Y 330.735,Z 416.046,A -85,B 0,C 180,E1 -15070.47,E2 -15070.47} C_VEL
LIN {X 0,Y 329.565,Z 410.167,A -85,B 0,C 180,E1 -15071.836,E2 -15071.836} C_VEL
LIN {X 0,Y 329.974,Z 406.182,A -85,B 0,C 180,E1 -15072.589,E2 -15072.589} C_VEL
LIN {X 0,Y 332.66,Z 394.516,A -85,B 0,C 180,E1 -15074.412,E2 -15074.412} C_VEL
LIN {X 0,Y 335.384,Z 381.839,A -85,B 0,C 180,E1 -15076.03,E2 -15076.03} C_VEL
LIN {X 0,Y 337.896,Z 368.87,A -85,B 0,C 180,E1 -15077.372,E2 -15077.372} C_VEL
LIN {X 0,Y 340.074,Z 354.864,A -85,B 0,C 180,E1 -15078.551,E2 -15078.551} C_VEL
LIN {X 0,Y 342.029,Z 340.346,A -85,B 0,C 180,E1 -15079.488,E2 -15079.488} C_VEL
LIN {X 0,Y 343.418,Z 327.372,A -85,B 0,C 180,E1 -15080.123,E2 -15080.123} C_VEL
LIN {X 0,Y 344.564,Z 312.542,A -85,B 0,C 180,E1 -15080.634,E2 -15080.634} C_VEL
LIN {X 0,Y 348.925,Z 199.288,A -85,B 0,C 180,E1 -15083.095,E2 -15083.095} C_VEL
LIN {X 0,Y 341.987,Z 184.913,A -85,B 0,C 180,E1 -15084.453,E2 -15084.453} C_VEL
LIN {X 0,Y 333.749,Z 170.186,A -85,B 0,C 180,E1 -15086.119,E2 -15086.119} C_VEL
LIN {X 0,Y 326.23,Z 158.099,A -85,B 0,C 180,E1 -15087.732,E2 -15087.732} C_VEL
LIN {X 0,Y 320.429,Z 149.252,A -85,B 0,C 180,E1 -15089.078,E2 -15089.078} C_VEL
LIN {X 0,Y 319.58,Z 146.298,A -85,B 0,C 180,E1 -15090.252,E2 -15090.252} C_VEL
LIN {X 0,Y 319.595,Z 146.295,A -85,B 0,C 180,E1 -15094.369,E2 -15094.369} C_VEL
LIN {X 0,Y 319.57,Z 146.303,A -85,B 0,C 180,E1 -15098.045,E2 -15098.045} C_VEL
LIN {X 0,Y 319.658,Z 146.293,A -85,B 0,C 180,E1 -15100.978,E2 -15100.978} C_VEL
LIN {X 0,Y 319.713,Z 146.279,A -85,B 0,C 180,E1 -15105.288,E2 -15105.288} C_VEL
LIN {X 0,Y 319.723,Z 146.279,A -85,B 0,C 180,E1 -15108.589,E2 -15108.589} C_VEL
LIN {X 0,Y 319.933,Z 146.258,A -85,B 0,C 180,E1 -15112.426,E2 -15112.426} C_VEL
LIN {X 0,Y 319.745,Z 146.273,A -85,B 0,C 180,E1 -15114.955,E2 -15114.955} C_VEL
LIN {X 0,Y 319.989,Z 146.244,A -85,B 0,C 180,E1 -15117.482,E2 -15117.482} C_VEL
LIN {X 0,Y 320.149,Z 146.231,A -85,B 0,C 180,E1 -15119.999,E2 -15119.999} C_VEL
LIN {X 0,Y 319.989,Z 146.247,A -85,B 0,C 180,E1 -15122.517,E2 -15122.517} C_VEL
LIN {X 0,Y 319.906,Z 146.259,A -85,B 0,C 180,E1 -15126.306,E2 -15126.306} C_VEL
LIN {X 0,Y 319.734,Z 146.281,A -85,B 0,C 180,E1 -15130.127,E2 -15130.127} C_VEL
LIN {X 0,Y 319.731,Z 146.282,A -85,B 0,C 180,E1 -15133.992,E2 -15133.992} C_VEL
LIN {X 0,Y 319.658,Z 146.292,A -85,B 0,C 180,E1 -15137.926,E2 -15137.926} C_VEL
LIN {X 0,Y 319.616,Z 146.293,A -85,B 0,C 180,E1 -15140.598,E2 -15140.598} C_VEL
LIN {X 0,Y 319.569,Z 146.297,A -85,B 0,C 180,E1 -15143.319,E2 -15143.319} C_VEL
LIN {X 0,Y 319.633,Z 146.288,A -85,B 0,C 180,E1 -15146.088,E2 -15146.088} C_VEL
LIN {X 0,Y 319.587,Z 146.295,A -85,B 0,C 180,E1 -15148.933,E2 -15148.933} C_VEL
LIN {X 0,Y 319.53,Z 146.303,A -85,B 0,C 180,E1 -15151.861,E2 -15151.861} C_VEL
LIN {X 0,Y 319.577,Z 146.299,A -85,B 0,C 180,E1 -15155.543,E2 -15155.543} C_VEL
LIN {X 0,Y 319.556,Z 146.288,A -85,B 0,C 180,E1 -15159.669,E2 -15159.669} C_VEL
LIN {X 0,Y 319.555,Z 146.288,A -85,B 0,C 180,E1 -15163.467,E2 -15163.467} C_VEL
LIN {X 0,Y 319.537,Z 146.384,A -85,B 0,C 180,E1 -15165.266,E2 -15165.266} C_VEL
LIN {X 0,Y 322.738,Z 156.002,A -85,B 0,C 180,E1 -15168.811,E2 -15168.811} C_VEL
LIN {X 0,Y 324.557,Z 161.781,A -85,B 0,C 180,E1 -15170.75,E2 -15170.75} C_VEL
LIN {X 0,Y 331.261,Z 173.187,A -85,B 0,C 180,E1 -15172.228,E2 -15172.228} C_VEL
LIN {X 0,Y 338.287,Z 186.023,A -85,B 0,C 180,E1 -15173.696,E2 -15173.696} C_VEL
LIN {X 0,Y 346.242,Z 202.586,A -85,B 0,C 180,E1 -15175.288,E2 -15175.288} C_VEL
LIN {X 0,Y 348.334,Z 214.275,A -85,B 0,C 180,E1 -15175.884,E2 -15175.884} C_VEL
LIN {X 0,Y 347.021,Z 252.279,A -85,B 0,C 180,E1 -15176.721,E2 -15176.721} C_VEL
LIN {X 0,Y 344.037,Z 329.01,A -85,B 0,C 180,E1 -15178.392,E2 -15178.392} C_VEL
LIN {X 0,Y 342.681,Z 344.755,A -85,B 0,C 180,E1 -15178.941,E2 -15178.941} C_VEL
LIN {X 0,Y 340.661,Z 360.39,A -85,B 0,C 180,E1 -15179.725,E2 -15179.725} C_VEL
LIN {X 0,Y 338.533,Z 374.789,A -85,B 0,C 180,E1 -15180.717,E2 -15180.717} C_VEL
LIN {X 0,Y 336.352,Z 387.143,A -85,B 0,C 180,E1 -15181.788,E2 -15181.788} C_VEL
LIN {X 0,Y 333.59,Z 400.721,A -85,B 0,C 180,E1 -15183.236,E2 -15183.236} C_VEL
LIN {X 0,Y 331.078,Z 411.995,A -85,B 0,C 180,E1 -15184.71,E2 -15184.71} C_VEL
LIN {X 0,Y 328.574,Z 422.552,A -85,B 0,C 180,E1 -15186.357,E2 -15186.357} C_VEL
LIN {X 0,Y 326.164,Z 432.484,A -85,B 0,C 180,E1 -15188.206,E2 -15188.206} C_VEL
LIN {X 0,Y 323.824,Z 442.03,A -85,B 0,C 180,E1 -15190.343,E2 -15190.343} C_VEL
LIN {X 0,Y 321.927,Z 450.121,A -85,B 0,C 180,E1 -15192.532,E2 -15192.532} C_VEL
LIN {X 0,Y 320.006,Z 458.269,A -85,B 0,C 180,E1 -15195.273,E2 -15195.273} C_VEL
LIN {X 0,Y 318.937,Z 464.407,A -85,B 0,C 180,E1 -15197.917,E2 -15197.917} C_VEL
LIN {X 0,Y 318.352,Z 467.924,A -85,B 0,C 180,E1 -15199.828,E2 -15199.828} C_VEL
LIN {X 0,Y 317.917,Z 471.526,A -85,B 0,C 180,E1 -15202.378,E2 -15202.378} C_VEL
LIN {X 0,Y 317.754,Z 473.942,A -85,B 0,C 180,E1 -15204.925,E2 -15204.925} C_VEL
LIN {X 0,Y 317.741,Z 475.212,A -85,B 0,C 180,E1 -15207.465,E2 -15207.465} C_VEL
LIN {X 0,Y 317.78,Z 475.283,A -85,B 0,C 180,E1 -15210.001,E2 -15210.001} C_VEL
LIN {X 0,Y 317.747,Z 474.195,A -85,B 0,C 180,E1 -15212.536,E2 -15212.536} C_VEL
LIN {X 0,Y 317.769,Z 471.933,A -85,B 0,C 180,E1 -15215.076,E2 -15215.076} C_VEL
LIN {X 0,Y 317.954,Z 468.443,A -85,B 0,C 180,E1 -15217.622,E2 -15217.622} C_VEL
LIN {X 0,Y 318.236,Z 463.619,A -85,B 0,C 180,E1 -15220.177,E2 -15220.177} C_VEL
LIN {X 0,Y 318.948,Z 457.34,A -85,B 0,C 180,E1 -15222.73,E2 -15222.73} C_VEL
LIN {X 0,Y 319.983,Z 449.415,A -85,B 0,C 180,E1 -15225.282,E2 -15225.282} C_VEL
LIN {X 0,Y 321.301,Z 440.962,A -85,B 0,C 180,E1 -15227.504,E2 -15227.504} C_VEL
LIN {X 0,Y 323.081,Z 430.749,A -85,B 0,C 180,E1 -15229.705,E2 -15229.705} C_VEL
LIN {X 0,Y 324.762,Z 420.282,A -85,B 0,C 180,E1 -15231.586,E2 -15231.586} C_VEL
LIN {X 0,Y 326.901,Z 407.739,A -85,B 0,C 180,E1 -15233.437,E2 -15233.437} C_VEL
LIN {X 0,Y 328.799,Z 395.133,A -85,B 0,C 180,E1 -15234.971,E2 -15234.971} C_VEL
LIN {X 0,Y 330.882,Z 381.336,A -85,B 0,C 180,E1 -15236.321,E2 -15236.321} C_VEL
LIN {X 0,Y 332.541,Z 368.034,A -85,B 0,C 180,E1 -15237.369,E2 -15237.369} C_VEL
LIN {X 0,Y 333.987,Z 353.563,A -85,B 0,C 180,E1 -15238.26,E2 -15238.26} C_VEL
LIN {X 0,Y 335.332,Z 337.959,A -85,B 0,C 180,E1 -15238.948,E2 -15238.948} C_VEL
LIN {X 0,Y 336.085,Z 322.678,A -85,B 0,C 180,E1 -15239.391,E2 -15239.391} C_VEL
LIN {X 0,Y 339.32,Z 212.314,A -85,B 0,C 180,E1 -15241.747,E2 -15241.747} C_VEL
LIN {X 0,Y 335.526,Z 190.627,A -85,B 0,C 180,E1 -15242.606,E2 -15242.606} C_VEL
LIN {X 0,Y 326.548,Z 169.256,A -85,B 0,C 180,E1 -15243.978,E2 -15243.978} C_VEL
LIN {X 0,Y 323.84,Z 162.844,A -85,B 0,C 180,E1 -15244.445,E2 -15244.445} C_VEL
LIN {X 0,Y 320.919,Z 151.305,A -85,B 0,C 180,E1 -15247.453,E2 -15247.453} C_VEL
LIN {X 0,Y 319.603,Z 146.298,A -85,B 0,C 180,E1 -15248.809,E2 -15248.809} C_VEL
LIN {X 0,Y 319.555,Z 146.306,A -85,B 0,C 180,E1 -15252.984,E2 -15252.984} C_VEL
LIN {X 0,Y 319.556,Z 146.31,A -85,B 0,C 180,E1 -15257.017,E2 -15257.017} C_VEL
LIN {X 0,Y 319.549,Z 146.298,A -85,B 0,C 180,E1 -15260.372,E2 -15260.372} C_VEL
LIN {X 0,Y 319.582,Z 146.298,A -85,B 0,C 180,E1 -15264.458,E2 -15264.458} C_VEL
LIN {X 0,Y 319.527,Z 146.306,A -85,B 0,C 180,E1 -15268.138,E2 -15268.138} C_VEL
LIN {X 0,Y 319.573,Z 146.279,A -85,B 0,C 180,E1 -15271.604,E2 -15271.604} C_VEL
LIN {X 0,Y 319.578,Z 146.3,A -85,B 0,C 180,E1 -15275.302,E2 -15275.302} C_VEL
LIN {X 0,Y 319.571,Z 146.295,A -85,B 0,C 180,E1 -15278.046,E2 -15278.046} C_VEL
LIN {X 0,Y 319.66,Z 146.291,A -85,B 0,C 180,E1 -15280.98,E2 -15280.98} C_VEL
LIN {X 0,Y 319.716,Z 146.284,A -85,B 0,C 180,E1 -15285.29,E2 -15285.29} C_VEL
LIN {X 0,Y 319.719,Z 146.28,A -85,B 0,C 180,E1 -15288.59,E2 -15288.59} C_VEL
LIN {X 0,Y 319.857,Z 146.261,A -85,B 0,C 180,E1 -15292.425,E2 -15292.425} C_VEL
LIN {X 0,Y 319.721,Z 146.282,A -85,B 0,C 180,E1 -15294.956,E2 -15294.956} C_VEL
LIN {X 0,Y 319.959,Z 146.24,A -85,B 0,C 180,E1 -15297.483,E2 -15297.483} C_VEL
LIN {X 0,Y 320.002,Z 146.23,A -85,B 0,C 180,E1 -15301.259,E2 -15301.259} C_VEL
LIN {X 0,Y 319.718,Z 146.281,A -85,B 0,C 180,E1 -15305.045,E2 -15305.045} C_VEL
LIN {X 0,Y 319.858,Z 146.247,A -85,B 0,C 180,E1 -15307.576,E2 -15307.576} C_VEL
LIN {X 0,Y 319.708,Z 146.265,A -85,B 0,C 180,E1 -15311.411,E2 -15311.411} C_VEL
LIN {X 0,Y 319.654,Z 146.29,A -85,B 0,C 180,E1 -15314.668,E2 -15314.668} C_VEL
LIN {X 0,Y 319.602,Z 146.296,A -85,B 0,C 180,E1 -15318.99,E2 -15318.99} C_VEL
LIN {X 0,Y 319.525,Z 146.305,A -85,B 0,C 180,E1 -15323.324,E2 -15323.324} C_VEL
LIN {X 0,Y 319.554,Z 146.299,A -85,B 0,C 180,E1 -15326.096,E2 -15326.096} C_VEL
LIN {X 0,Y 319.526,Z 146.278,A -85,B 0,C 180,E1 -15328.941,E2 -15328.941} C_VEL
LIN {X 0,Y 319.528,Z 146.299,A -85,B 0,C 180,E1 -15331.863,E2 -15331.863} C_VEL
LIN {X 0,Y 319.583,Z 146.294,A -85,B 0,C 180,E1 -15335.542,E2 -15335.542} C_VEL
LIN {X 0,Y 319.533,Z 146.291,A -85,B 0,C 180,E1 -15339.662,E2 -15339.662} C_VEL
LIN {X 0,Y 319.524,Z 146.303,A -85,B 0,C 180,E1 -15343.46,E2 -15343.46} C_VEL
LIN {X 0,Y 319.556,Z 146.289,A -85,B 0,C 180,E1 -15347.016,E2 -15347.016} C_VEL
LIN {X 0,Y 319.519,Z 146.307,A -85,B 0,C 180,E1 -15350.366,E2 -15350.366} C_VEL
LIN {X 0,Y 319.585,Z 146.3,A -85,B 0,C 180,E1 -15354.457,E2 -15354.457} C_VEL
LIN {X 0,Y 319.529,Z 146.298,A -85,B 0,C 180,E1 -15358.137,E2 -15358.137} C_VEL
LIN {X 0,Y 319.576,Z 146.296,A -85,B 0,C 180,E1 -15361.604,E2 -15361.604} C_VEL
LIN {X 0,Y 319.547,Z 146.309,A -85,B 0,C 180,E1 -15365.299,E2 -15365.299} C_VEL
LIN {X 0,Y 319.57,Z 146.305,A -85,B 0,C 180,E1 -15368.045,E2 -15368.045} C_VEL
LIN {X 0,Y 319.663,Z 146.281,A -85,B 0,C 180,E1 -15370.978,E2 -15370.978} C_VEL
LIN {X 0,Y 319.696,Z 146.317,A -85,B 0,C 180,E1 -15373.837,E2 -15373.837} C_VEL
LIN {X 0,Y 320.192,Z 148.126,A -85,B 0,C 180,E1 -15374.311,E2 -15374.311} C_VEL
LIN {X 0,Y 330.18,Z 169.468,A -85,B 0,C 180,E1 -15375.844,E2 -15375.844} C_VEL
LIN {X 0,Y 339.671,Z 192.12,A -85,B 0,C 180,E1 -15377.267,E2 -15377.267} C_VEL
LIN {X 0,Y 338.038,Z 251.542,A -85,B 0,C 180,E1 -15378.544,E2 -15378.544} C_VEL
LIN {X 0,Y 336.126,Z 313.474,A -85,B 0,C 180,E1 -15379.901,E2 -15379.901} C_VEL
LIN {X 0,Y 335.199,Z 328.57,A -85,B 0,C 180,E1 -15380.458,E2 -15380.458} C_VEL
LIN {X 0,Y 334.026,Z 342.584,A -85,B 0,C 180,E1 -15381.195,E2 -15381.195} C_VEL
LIN {X 0,Y 332.348,Z 357.782,A -85,B 0,C 180,E1 -15382.252,E2 -15382.252} C_VEL
LIN {X 0,Y 330.687,Z 371.084,A -85,B 0,C 180,E1 -15383.44,E2 -15383.44} C_VEL
LIN {X 0,Y 328.657,Z 384.707,A -85,B 0,C 180,E1 -15384.939,E2 -15384.939} C_VEL
LIN {X 0,Y 326.672,Z 397.038,A -85,B 0,C 180,E1 -15386.608,E2 -15386.608} C_VEL
LIN {X 0,Y 324.808,Z 408.265,A -85,B 0,C 180,E1 -15388.45,E2 -15388.45} C_VEL
LIN {X 0,Y 322.956,Z 419.197,A -85,B 0,C 180,E1 -15390.622,E2 -15390.622} C_VEL
LIN {X 0,Y 321.342,Z 428.299,A -85,B 0,C 180,E1 -15392.82,E2 -15392.82} C_VEL
LIN {X 0,Y 320.15,Z 435.837,A -85,B 0,C 180,E1 -15395.037,E2 -15395.037} C_VEL
LIN {X 0,Y 319.109,Z 443.061,A -85,B 0,C 180,E1 -15397.657,E2 -15397.657} C_VEL
LIN {X 0,Y 318.396,Z 448.452,A -85,B 0,C 180,E1 -15400.17,E2 -15400.17} C_VEL
LIN {X 0,Y 317.931,Z 452.636,A -85,B 0,C 180,E1 -15402.77,E2 -15402.77} C_VEL
LIN {X 0,Y 317.613,Z 455.544,A -85,B 0,C 180,E1 -15405.398,E2 -15405.398} C_VEL
LIN {X 0,Y 317.568,Z 457.205,A -85,B 0,C 180,E1 -15408.049,E2 -15408.049} C_VEL
LIN {X 0,Y 317.582,Z 457.628,A -85,B 0,C 180,E1 -15410.736,E2 -15410.736} C_VEL
LIN {X 0,Y 317.753,Z 456.773,A -85,B 0,C 180,E1 -15413.46,E2 -15413.46} C_VEL
LIN {X 0,Y 318.223,Z 454.582,A -85,B 0,C 180,E1 -15416.212,E2 -15416.212} C_VEL
LIN {X 0,Y 318.974,Z 450.961,A -85,B 0,C 180,E1 -15418.994,E2 -15418.994} C_VEL
LIN {X 0,Y 320.099,Z 445.782,A -85,B 0,C 180,E1 -15421.798,E2 -15421.798} C_VEL
LIN {X 0,Y 321.473,Z 440.253,A -85,B 0,C 180,E1 -15424.112,E2 -15424.112} C_VEL
LIN {X 0,Y 323.18,Z 433.365,A -85,B 0,C 180,E1 -15426.426,E2 -15426.426} C_VEL
LIN {X 0,Y 325.369,Z 424.721,A -85,B 0,C 180,E1 -15428.785,E2 -15428.785} C_VEL
LIN {X 0,Y 327.673,Z 415.465,A -85,B 0,C 180,E1 -15430.856,E2 -15430.856} C_VEL
LIN {X 0,Y 329.974,Z 406.182,A -85,B 0,C 180,E1 -15432.589,E2 -15432.589} C_VEL
LIN {X 0,Y 330.431,Z 402.121,A -85,B 0,C 180,E1 -15433.327,E2 -15433.327} C_VEL
LIN {X 0,Y 329.519,Z 395.508,A -85,B 0,C 180,E1 -15434.603,E2 -15434.603} C_VEL
LIN {X 0,Y 328.57,Z 388.562,A -85,B 0,C 180,E1 -15435.822,E2 -15435.822} C_VEL
LIN {X 0,Y 328.942,Z 383.938,A -85,B 0,C 180,E1 -15436.457,E2 -15436.457} C_VEL
LIN {X 0,Y 331.358,Z 372.269,A -85,B 0,C 180,E1 -15437.738,E2 -15437.738} C_VEL
LIN {X 0,Y 333.698,Z 358.676,A -85,B 0,C 180,E1 -15438.959,E2 -15438.959} C_VEL
LIN {X 0,Y 335.825,Z 344.264,A -85,B 0,C 180,E1 -15439.968,E2 -15439.968} C_VEL
LIN {X 0,Y 337.422,Z 330.175,A -85,B 0,C 180,E1 -15440.717,E2 -15440.717} C_VEL
LIN {X 0,Y 338.694,Z 315.464,A -85,B 0,C 180,E1 -15441.266,E2 -15441.266} C_VEL
LIN {X 0,Y 339.706,Z 292.075,A -85,B 0,C 180,E1 -15441.828,E2 -15441.828} C_VEL
LIN {X 0,Y 343.406,Z 201.675,A -85,B 0,C 180,E1 -15443.787,E2 -15443.787} C_VEL
LIN {X 0,Y 336.266,Z 187.041,A -85,B 0,C 180,E1 -15445.236,E2 -15445.236} C_VEL
LIN {X 0,Y 327.903,Z 172.171,A -85,B 0,C 180,E1 -15447.014,E2 -15447.014} C_VEL
LIN {X 0,Y 321.143,Z 161.499,A -85,B 0,C 180,E1 -15448.521,E2 -15448.521} C_VEL
LIN {X 0,Y 315.984,Z 153.817,A -85,B 0,C 180,E1 -15449.74,E2 -15449.74} C_VEL
LIN {X 0,Y 313.642,Z 150.219,A -85,B 0,C 180,E1 -15450.325,E2 -15450.325} C_VEL
LIN {X 0,Y 313.313,Z 149.582,A -85,B 0,C 180,E1 -15450.429,E2 -15450.429} C_VEL
LIN {X 0,Y 312.544,Z 147.161,A -85,B 0,C 180,E1 -15451.51,E2 -15451.51} C_VEL
LIN {X 0,Y 312.555,Z 147.165,A -85,B 0,C 180,E1 -15454.708,E2 -15454.708} C_VEL
LIN {X 0,Y 312.566,Z 147.167,A -85,B 0,C 180,E1 -15457.527,E2 -15457.527} C_VEL
LIN {X 0,Y 312.589,Z 147.169,A -85,B 0,C 180,E1 -15461.653,E2 -15461.653} C_VEL
LIN {X 0,Y 312.686,Z 147.156,A -85,B 0,C 180,E1 -15465.685,E2 -15465.685} C_VEL
LIN {X 0,Y 312.702,Z 147.161,A -85,B 0,C 180,E1 -15469.641,E2 -15469.641} C_VEL
LIN {X 0,Y 312.872,Z 147.136,A -85,B 0,C 180,E1 -15472.254,E2 -15472.254} C_VEL
LIN {X 0,Y 312.715,Z 147.148,A -85,B 0,C 180,E1 -15474.842,E2 -15474.842} C_VEL
LIN {X 0,Y 312.988,Z 147.116,A -85,B 0,C 180,E1 -15478.713,E2 -15478.713} C_VEL
LIN {X 0,Y 312.988,Z 147.115,A -85,B 0,C 180,E1 -15481.286,E2 -15481.286} C_VEL
LIN {X 0,Y 312.705,Z 147.15,A -85,B 0,C 180,E1 -15485.157,E2 -15485.157} C_VEL
LIN {X 0,Y 312.798,Z 147.144,A -85,B 0,C 180,E1 -15487.747,E2 -15487.747} C_VEL
LIN {X 0,Y 312.663,Z 147.159,A -85,B 0,C 180,E1 -15491.671,E2 -15491.671} C_VEL
LIN {X 0,Y 312.699,Z 147.157,A -85,B 0,C 180,E1 -15494.887,E2 -15494.887} C_VEL
LIN {X 0,Y 312.63,Z 147.159,A -85,B 0,C 180,E1 -15499.237,E2 -15499.237} C_VEL
LIN {X 0,Y 312.544,Z 147.171,A -85,B 0,C 180,E1 -15502.789,E2 -15502.789} C_VEL
LIN {X 0,Y 312.601,Z 147.165,A -85,B 0,C 180,E1 -15505.935,E2 -15505.935} C_VEL
LIN {X 0,Y 312.543,Z 147.172,A -85,B 0,C 180,E1 -15509.65,E2 -15509.65} C_VEL
LIN {X 0,Y 312.517,Z 147.183,A -85,B 0,C 180,E1 -15513.689,E2 -15513.689} C_VEL
LIN {X 0,Y 312.518,Z 147.169,A -85,B 0,C 180,E1 -15517.386,E2 -15517.386} C_VEL
LIN {X 0,Y 312.488,Z 147.185,A -85,B 0,C 180,E1 -15520.709,E2 -15520.709} C_VEL
LIN {X 0,Y 312.48,Z 147.237,A -85,B 0,C 180,E1 -15524.034,E2 -15524.034} C_VEL
LIN {X 0,Y 315.629,Z 156.555,A -85,B 0,C 180,E1 -15527.669,E2 -15527.669} C_VEL
LIN {X 0,Y 317.265,Z 161.511,A -85,B 0,C 180,E1 -15529.423,E2 -15529.423} C_VEL
LIN {X 0,Y 319.942,Z 166.047,A -85,B 0,C 180,E1 -15530.065,E2 -15530.065} C_VEL
LIN {X 0,Y 324.656,Z 173.819,A -85,B 0,C 180,E1 -15531.144,E2 -15531.144} C_VEL
LIN {X 0,Y 331.607,Z 186.21,A -85,B 0,C 180,E1 -15532.673,E2 -15532.673} C_VEL
LIN {X 0,Y 340.051,Z 203.441,A -85,B 0,C 180,E1 -15534.444,E2 -15534.444} C_VEL
LIN {X 0,Y 341.335,Z 206.809,A -85,B 0,C 180,E1 -15534.721,E2 -15534.721} C_VEL
LIN {X 0,Y 342.864,Z 216.506,A -85,B 0,C 180,E1 -15535.202,E2 -15535.202} C_VEL
LIN {X 0,Y 338.38,Z 328.379,A -85,B 0,C 180,E1 -15537.669,E2 -15537.669} C_VEL
LIN {X 0,Y 337.062,Z 343.411,A -85,B 0,C 180,E1 -15538.188,E2 -15538.188} C_VEL
LIN {X 0,Y 335.133,Z 358.163,A -85,B 0,C 180,E1 -15538.909,E2 -15538.909} C_VEL
LIN {X 0,Y 333.099,Z 371.992,A -85,B 0,C 180,E1 -15539.839,E2 -15539.839} C_VEL
LIN {X 0,Y 330.71,Z 384.85,A -85,B 0,C 180,E1 -15540.914,E2 -15540.914} C_VEL
LIN {X 0,Y 327.886,Z 398.801,A -85,B 0,C 180,E1 -15542.386,E2 -15542.386} C_VEL
LIN {X 0,Y 325.155,Z 410.374,A -85,B 0,C 180,E1 -15543.872,E2 -15543.872} C_VEL
LIN {X 0,Y 322.551,Z 421.162,A -85,B 0,C 180,E1 -15545.545,E2 -15545.545} C_VEL
LIN {X 0,Y 319.776,Z 431.85,A -85,B 0,C 180,E1 -15547.537,E2 -15547.537} C_VEL
LIN {X 0,Y 317.471,Z 440.984,A -85,B 0,C 180,E1 -15549.595,E2 -15549.595} C_VEL
LIN {X 0,Y 315.126,Z 450.222,A -85,B 0,C 180,E1 -15552.143,E2 -15552.143} C_VEL
LIN {X 0,Y 313.144,Z 457.986,A -85,B 0,C 180,E1 -15554.809,E2 -15554.809} C_VEL
LIN {X 0,Y 311.956,Z 464.392,A -85,B 0,C 180,E1 -15557.642,E2 -15557.642} C_VEL
LIN {X 0,Y 311.312,Z 467.884,A -85,B 0,C 180,E1 -15559.596,E2 -15559.596} C_VEL
LIN {X 0,Y 310.834,Z 471.434,A -85,B 0,C 180,E1 -15562.204,E2 -15562.204} C_VEL
LIN {X 0,Y 310.682,Z 473.801,A -85,B 0,C 180,E1 -15564.809,E2 -15564.809} C_VEL
LIN {X 0,Y 310.663,Z 475.026,A -85,B 0,C 180,E1 -15567.407,E2 -15567.407} C_VEL
LIN {X 0,Y 310.69,Z 475.072,A -85,B 0,C 180,E1 -15570.001,E2 -15570.001} C_VEL
LIN {X 0,Y 310.67,Z 473.939,A -85,B 0,C 180,E1 -15572.594,E2 -15572.594} C_VEL
LIN {X 0,Y 310.682,Z 471.63,A -85,B 0,C 180,E1 -15575.192,E2 -15575.192} C_VEL
LIN {X 0,Y 310.878,Z 468.089,A -85,B 0,C 180,E1 -15577.796,E2 -15577.796} C_VEL
LIN {X 0,Y 311.169,Z 463.208,A -85,B 0,C 180,E1 -15580.41,E2 -15580.41} C_VEL
LIN {X 0,Y 311.937,Z 456.867,A -85,B 0,C 180,E1 -15583.021,E2 -15583.021} C_VEL
LIN {X 0,Y 313.046,Z 448.87,A -85,B 0,C 180,E1 -15585.629,E2 -15585.629} C_VEL
LIN {X 0,Y 314.422,Z 440.334,A -85,B 0,C 180,E1 -15587.9,E2 -15587.9} C_VEL
LIN {X 0,Y 316.018,Z 431.65,A -85,B 0,C 180,E1 -15589.826,E2 -15589.826} C_VEL
LIN {X 0,Y 317.887,Z 420.524,A -85,B 0,C 180,E1 -15591.89,E2 -15591.89} C_VEL
LIN {X 0,Y 320.105,Z 407.984,A -85,B 0,C 180,E1 -15593.793,E2 -15593.793} C_VEL
LIN {X 0,Y 322.061,Z 395.456,A -85,B 0,C 180,E1 -15595.358,E2 -15595.358} C_VEL
LIN {X 0,Y 324.223,Z 381.789,A -85,B 0,C 180,E1 -15596.731,E2 -15596.731} C_VEL
LIN {X 0,Y 325.954,Z 368.252,A -85,B 0,C 180,E1 -15597.825,E2 -15597.825} C_VEL
LIN {X 0,Y 327.561,Z 353.043,A -85,B 0,C 180,E1 -15598.778,E2 -15598.778} C_VEL
LIN {X 0,Y 328.92,Z 337.276,A -85,B 0,C 180,E1 -15599.48,E2 -15599.48} C_VEL
LIN {X 0,Y 329.714,Z 321.702,A -85,B 0,C 180,E1 -15599.929,E2 -15599.929} C_VEL
LIN {X 0,Y 332.999,Z 213.187,A -85,B 0,C 180,E1 -15602.285,E2 -15602.285} C_VEL
LIN {X 0,Y 329.52,Z 193.283,A -85,B 0,C 180,E1 -15603.093,E2 -15603.093} C_VEL
LIN {X 0,Y 321.098,Z 173.005,A -85,B 0,C 180,E1 -15604.423,E2 -15604.423} C_VEL
LIN {X 0,Y 316.523,Z 162.683,A -85,B 0,C 180,E1 -15605.187,E2 -15605.187} C_VEL
LIN {X 0,Y 313.556,Z 151.008,A -85,B 0,C 180,E1 -15608.328,E2 -15608.328} C_VEL
LIN {X 0,Y 312.52,Z 147.184,A -85,B 0,C 180,E1 -15609.426,E2 -15609.426} C_VEL
LIN {X 0,Y 312.491,Z 147.185,A -85,B 0,C 180,E1 -15612.432,E2 -15612.432} C_VEL
LIN {X 0,Y 312.46,Z 147.193,A -85,B 0,C 180,E1 -15616.036,E2 -15616.036} C_VEL
LIN {X 0,Y 312.506,Z 147.179,A -85,B 0,C 180,E1 -15619.875,E2 -15619.875} C_VEL
LIN {X 0,Y 312.537,Z 147.176,A -85,B 0,C 180,E1 -15624.051,E2 -15624.051} C_VEL
LIN {X 0,Y 312.504,Z 147.18,A -85,B 0,C 180,E1 -15627.334,E2 -15627.334} C_VEL
LIN {X 0,Y 312.509,Z 147.161,A -85,B 0,C 180,E1 -15631.292,E2 -15631.292} C_VEL
LIN {X 0,Y 312.55,Z 147.168,A -85,B 0,C 180,E1 -15634.708,E2 -15634.708} C_VEL
LIN {X 0,Y 312.567,Z 147.168,A -85,B 0,C 180,E1 -15637.528,E2 -15637.528} C_VEL
LIN {X 0,Y 312.592,Z 147.168,A -85,B 0,C 180,E1 -15641.654,E2 -15641.654} C_VEL
LIN {X 0,Y 312.689,Z 147.159,A -85,B 0,C 180,E1 -15645.686,E2 -15645.686} C_VEL
LIN {X 0,Y 312.69,Z 147.158,A -85,B 0,C 180,E1 -15649.642,E2 -15649.642} C_VEL
LIN {X 0,Y 312.8,Z 147.14,A -85,B 0,C 180,E1 -15652.253,E2 -15652.253} C_VEL
LIN {X 0,Y 312.692,Z 147.159,A -85,B 0,C 180,E1 -15654.842,E2 -15654.842} C_VEL
LIN {X 0,Y 312.971,Z 147.093,A -85,B 0,C 180,E1 -15658.714,E2 -15658.714} C_VEL
LIN {X 0,Y 312.97,Z 147.106,A -85,B 0,C 180,E1 -15661.287,E2 -15661.287} C_VEL
LIN {X 0,Y 312.689,Z 147.157,A -85,B 0,C 180,E1 -15665.159,E2 -15665.159} C_VEL
LIN {X 0,Y 312.801,Z 147.122,A -85,B 0,C 180,E1 -15667.748,E2 -15667.748} C_VEL
LIN {X 0,Y 312.655,Z 147.145,A -85,B 0,C 180,E1 -15671.672,E2 -15671.672} C_VEL
LIN {X 0,Y 312.607,Z 147.168,A -85,B 0,C 180,E1 -15674.82,E2 -15674.82} C_VEL
LIN {X 0,Y 312.535,Z 147.178,A -85,B 0,C 180,E1 -15679.184,E2 -15679.184} C_VEL
LIN {X 0,Y 312.505,Z 147.175,A -85,B 0,C 180,E1 -15682.769,E2 -15682.769} C_VEL
LIN {X 0,Y 312.486,Z 147.178,A -85,B 0,C 180,E1 -15686.732,E2 -15686.732} C_VEL
LIN {X 0,Y 312.47,Z 147.155,A -85,B 0,C 180,E1 -15689.658,E2 -15689.658} C_VEL
LIN {X 0,Y 312.525,Z 147.179,A -85,B 0,C 180,E1 -15693.689,E2 -15693.689} C_VEL
LIN {X 0,Y 312.514,Z 147.156,A -85,B 0,C 180,E1 -15697.388,E2 -15697.388} C_VEL
LIN {X 0,Y 312.446,Z 147.182,A -85,B 0,C 180,E1 -15700.717,E2 -15700.717} C_VEL
LIN {X 0,Y 312.455,Z 147.18,A -85,B 0,C 180,E1 -15704.21,E2 -15704.21} C_VEL
LIN {X 0,Y 312.46,Z 147.183,A -85,B 0,C 180,E1 -15707.925,E2 -15707.925} C_VEL
LIN {X 0,Y 312.481,Z 147.171,A -85,B 0,C 180,E1 -15711.924,E2 -15711.924} C_VEL
LIN {X 0,Y 312.536,Z 147.176,A -85,B 0,C 180,E1 -15714.22,E2 -15714.22} C_VEL
LIN {X 0,Y 312.507,Z 147.17,A -85,B 0,C 180,E1 -15717.333,E2 -15717.333} C_VEL
LIN {X 0,Y 312.511,Z 147.177,A -85,B 0,C 180,E1 -15721.291,E2 -15721.291} C_VEL
LIN {X 0,Y 312.528,Z 147.183,A -85,B 0,C 180,E1 -15724.705,E2 -15724.705} C_VEL
LIN {X 0,Y 312.537,Z 147.179,A -85,B 0,C 180,E1 -15728.912,E2 -15728.912} C_VEL
LIN {X 0,Y 312.594,Z 147.153,A -85,B 0,C 180,E1 -15731.653,E2 -15731.653} C_VEL
LIN {X 0,Y 312.633,Z 147.256,A -85,B 0,C 180,E1 -15733.272,E2 -15733.272} C_VEL
LIN {X 0,Y 312.891,Z 148.316,A -85,B 0,C 180,E1 -15733.539,E2 -15733.539} C_VEL
LIN {X 0,Y 321.648,Z 166.488,A -85,B 0,C 180,E1 -15734.933,E2 -15734.933} C_VEL
LIN {X 0,Y 332.356,Z 191.337,A -85,B 0,C 180,E1 -15736.588,E2 -15736.588} C_VEL
LIN {X 0,Y 333.456,Z 194.295,A -85,B 0,C 180,E1 -15736.76,E2 -15736.76} C_VEL
LIN {X 0,Y 329.715,Z 313.313,A -85,B 0,C 180,E1 -15739.373,E2 -15739.373} C_VEL
LIN {X 0,Y 328.75,Z 328.857,A -85,B 0,C 180,E1 -15739.957,E2 -15739.957} C_VEL
LIN {X 0,Y 327.569,Z 342.362,A -85,B 0,C 180,E1 -15740.677,E2 -15740.677} C_VEL
LIN {X 0,Y 326.079,Z 356.068,A -85,B 0,C 180,E1 -15741.634,E2 -15741.634} C_VEL
LIN {X 0,Y 324.304,Z 369.755,A -85,B 0,C 180,E1 -15742.841,E2 -15742.841} C_VEL
LIN {X 0,Y 322.377,Z 382.378,A -85,B 0,C 180,E1 -15744.213,E2 -15744.213} C_VEL
LIN {X 0,Y 320.495,Z 394.061,A -85,B 0,C 180,E1 -15745.755,E2 -15745.755} C_VEL
LIN {X 0,Y 318.654,Z 404.916,A -85,B 0,C 180,E1 -15747.471,E2 -15747.471} C_VEL
LIN {X 0,Y 316.883,Z 414.75,A -85,B 0,C 180,E1 -15749.316,E2 -15749.316} C_VEL
LIN {X 0,Y 315.32,Z 423.512,A -85,B 0,C 180,E1 -15751.277,E2 -15751.277} C_VEL
LIN {X 0,Y 313.874,Z 431.893,A -85,B 0,C 180,E1 -15753.53,E2 -15753.53} C_VEL
LIN {X 0,Y 312.696,Z 438.87,A -85,B 0,C 180,E1 -15755.804,E2 -15755.804} C_VEL
LIN {X 0,Y 311.744,Z 445.347,A -85,B 0,C 180,E1 -15758.426,E2 -15758.426} C_VEL
LIN {X 0,Y 311.146,Z 450.373,A -85,B 0,C 180,E1 -15761.069,E2 -15761.069} C_VEL
LIN {X 0,Y 310.725,Z 453.75,A -85,B 0,C 180,E1 -15763.446,E2 -15763.446} C_VEL
LIN {X 0,Y 310.491,Z 456.048,A -85,B 0,C 180,E1 -15765.76,E2 -15765.76} C_VEL
LIN {X 0,Y 310.439,Z 457.541,A -85,B 0,C 180,E1 -15768.478,E2 -15768.478} C_VEL
LIN {X 0,Y 310.5,Z 457.791,A -85,B 0,C 180,E1 -15771.232,E2 -15771.232} C_VEL
LIN {X 0,Y 310.731,Z 456.76,A -85,B 0,C 180,E1 -15774.023,E2 -15774.023} C_VEL
LIN {X 0,Y 311.276,Z 454.385,A -85,B 0,C 180,E1 -15776.843,E2 -15776.843} C_VEL
LIN {X 0,Y 312.112,Z 450.567,A -85,B 0,C 180,E1 -15779.695,E2 -15779.695} C_VEL
LIN {X 0,Y 313.411,Z 445.182,A -85,B 0,C 180,E1 -15782.56,E2 -15782.56} C_VEL
LIN {X 0,Y 314.82,Z 439.909,A -85,B 0,C 180,E1 -15784.747,E2 -15784.747} C_VEL
LIN {X 0,Y 316.523,Z 433.499,A -85,B 0,C 180,E1 -15786.932,E2 -15786.932} C_VEL
LIN {X 0,Y 318.768,Z 425.119,A -85,B 0,C 180,E1 -15789.267,E2 -15789.267} C_VEL
LIN {X 0,Y 321.221,Z 415.843,A -85,B 0,C 180,E1 -15791.39,E2 -15791.39} C_VEL
LIN {X 0,Y 324.143,Z 404.589,A -85,B 0,C 180,E1 -15793.503,E2 -15793.503} C_VEL
LIN {X 0,Y 326.791,Z 393.522,A -85,B 0,C 180,E1 -15795.21,E2 -15795.21} C_VEL
LIN {X 0,Y 328.942,Z 383.938,A -85,B 0,C 180,E1 -15796.457,E2 -15796.457} C_VEL
LIN {X 0,Y 329.359,Z 379.233,A -85,B 0,C 180,E1 -15797.075,E2 -15797.075} C_VEL
LIN {X 0,Y 327.683,Z 365.299,A -85,B 0,C 180,E1 -15799.006,E2 -15799.006} C_VEL
LIN {X 0,Y 327.691,Z 360.279,A -85,B 0,C 180,E1 -15799.546,E2 -15799.546} C_VEL
LIN {X 0,Y 327.93,Z 358.533,A -85,B 0,C 180,E1 -15799.697,E2 -15799.697} C_VEL
LIN {X 0,Y 330.181,Z 343.756,A -85,B 0,C 180,E1 -15800.737,E2 -15800.737} C_VEL
LIN {X 0,Y 331.925,Z 328.983,A -85,B 0,C 180,E1 -15801.513,E2 -15801.513} C_VEL
LIN {X 0,Y 333.259,Z 313.429,A -85,B 0,C 180,E1 -15802.071,E2 -15802.071} C_VEL
LIN {X 0,Y 337.853,Z 203.922,A -85,B 0,C 180,E1 -15804.519,E2 -15804.519} C_VEL
LIN {X 0,Y 331.428,Z 190.818,A -85,B 0,C 180,E1 -15805.878,E2 -15805.878} C_VEL
LIN {X 0,Y 323.847,Z 177.168,A -85,B 0,C 180,E1 -15807.548,E2 -15807.548} C_VEL
LIN {X 0,Y 316.012,Z 164.567,A -85,B 0,C 180,E1 -15809.374,E2 -15809.374} C_VEL
LIN {X 0,Y 311.591,Z 158.233,A -85,B 0,C 180,E1 -15810.461,E2 -15810.461} C_VEL
LIN {X 0,Y 309.02,Z 154.327,A -85,B 0,C 180,E1 -15811.127,E2 -15811.127} C_VEL
LIN {X 0,Y 305.992,Z 149.885,A -85,B 0,C 180,E1 -15811.957,E2 -15811.957} C_VEL
LIN {X 0,Y 305.467,Z 148.047,A -85,B 0,C 180,E1 -15812.77,E2 -15812.77} C_VEL
LIN {X 0,Y 305.489,Z 148.036,A -85,B 0,C 180,E1 -15815.536,E2 -15815.536} C_VEL
LIN {X 0,Y 305.501,Z 148.051,A -85,B 0,C 180,E1 -15819.813,E2 -15819.813} C_VEL
LIN {X 0,Y 305.547,Z 148.045,A -85,B 0,C 180,E1 -15822.601,E2 -15822.601} C_VEL
LIN {X 0,Y 305.627,Z 148.033,A -85,B 0,C 180,E1 -15825.347,E2 -15825.347} C_VEL
LIN {X 0,Y 305.639,Z 148.038,A -85,B 0,C 180,E1 -15829.399,E2 -15829.399} C_VEL
LIN {X 0,Y 305.813,Z 148.013,A -85,B 0,C 180,E1 -15832.074,E2 -15832.074} C_VEL
LIN {X 0,Y 305.687,Z 148.023,A -85,B 0,C 180,E1 -15834.723,E2 -15834.723} C_VEL
LIN {X 0,Y 305.955,Z 147.992,A -85,B 0,C 180,E1 -15838.683,E2 -15838.683} C_VEL
LIN {X 0,Y 305.955,Z 147.991,A -85,B 0,C 180,E1 -15841.316,E2 -15841.316} C_VEL
LIN {X 0,Y 305.673,Z 148.025,A -85,B 0,C 180,E1 -15845.276,E2 -15845.276} C_VEL
LIN {X 0,Y 305.748,Z 148.021,A -85,B 0,C 180,E1 -15847.927,E2 -15847.927} C_VEL
LIN {X 0,Y 305.598,Z 148.037,A -85,B 0,C 180,E1 -15851.945,E2 -15851.945} C_VEL
LIN {X 0,Y 305.637,Z 148.035,A -85,B 0,C 180,E1 -15855.035,E2 -15855.035} C_VEL
LIN {X 0,Y 305.576,Z 148.037,A -85,B 0,C 180,E1 -15859.445,E2 -15859.445} C_VEL
LIN {X 0,Y 305.489,Z 148.049,A -85,B 0,C 180,E1 -15863.041,E2 -15863.041} C_VEL
LIN {X 0,Y 305.546,Z 148.043,A -85,B 0,C 180,E1 -15866.227,E2 -15866.227} C_VEL
LIN {X 0,Y 305.493,Z 148.05,A -85,B 0,C 180,E1 -15869.05,E2 -15869.05} C_VEL
LIN {X 0,Y 305.442,Z 148.057,A -85,B 0,C 180,E1 -15871.952,E2 -15871.952} C_VEL
LIN {X 0,Y 305.46,Z 148.056,A -85,B 0,C 180,E1 -15875.113,E2 -15875.113} C_VEL
LIN {X 0,Y 305.438,Z 148.04,A -85,B 0,C 180,E1 -15878.526,E2 -15878.526} C_VEL
LIN {X 0,Y 305.457,Z 148.044,A -85,B 0,C 180,E1 -15882.587,E2 -15882.587} C_VEL
LIN {X 0,Y 306.006,Z 150.129,A -85,B 0,C 180,E1 -15883.551,E2 -15883.551} C_VEL
LIN {X 0,Y 308.759,Z 157.939,A -85,B 0,C 180,E1 -15886.751,E2 -15886.751} C_VEL
LIN {X 0,Y 309.907,Z 161.309,A -85,B 0,C 180,E1 -15887.961,E2 -15887.961} C_VEL
LIN {X 0,Y 313.069,Z 166.215,A -85,B 0,C 180,E1 -15888.767,E2 -15888.767} C_VEL
LIN {X 0,Y 320.543,Z 178.687,A -85,B 0,C 180,E1 -15890.579,E2 -15890.579} C_VEL
LIN {X 0,Y 327.248,Z 190.808,A -85,B 0,C 180,E1 -15892.104,E2 -15892.104} C_VEL
LIN {X 0,Y 334.661,Z 206.105,A -85,B 0,C 180,E1 -15893.728,E2 -15893.728} C_VEL
LIN {X 0,Y 336.19,Z 209.869,A -85,B 0,C 180,E1 -15894.063,E2 -15894.063} C_VEL
LIN {X 0,Y 337.389,Z 217.005,A -85,B 0,C 180,E1 -15894.44,E2 -15894.44} C_VEL
LIN {X 0,Y 332.692,Z 329.203,A -85,B 0,C 180,E1 -15896.957,E2 -15896.957} C_VEL
LIN {X 0,Y 331.322,Z 343.94,A -85,B 0,C 180,E1 -15897.481,E2 -15897.481} C_VEL
LIN {X 0,Y 329.154,Z 359.678,A -85,B 0,C 180,E1 -15898.279,E2 -15898.279} C_VEL
LIN {X 0,Y 327.001,Z 373.359,A -85,B 0,C 180,E1 -15899.234,E2 -15899.234} C_VEL
LIN {X 0,Y 324.576,Z 385.716,A -85,B 0,C 180,E1 -15900.31,E2 -15900.31} C_VEL
LIN {X 0,Y 321.967,Z 398.172,A -85,B 0,C 180,E1 -15901.656,E2 -15901.656} C_VEL
LIN {X 0,Y 318.795,Z 410.87,A -85,B 0,C 180,E1 -15903.31,E2 -15903.31} C_VEL
LIN {X 0,Y 316.095,Z 421.543,A -85,B 0,C 180,E1 -15905.012,E2 -15905.012} C_VEL
LIN {X 0,Y 313.087,Z 432.579,A -85,B 0,C 180,E1 -15907.135,E2 -15907.135} C_VEL
LIN {X 0,Y 310.445,Z 442.414,A -85,B 0,C 180,E1 -15909.458,E2 -15909.458} C_VEL
LIN {X 0,Y 308.044,Z 451.359,A -85,B 0,C 180,E1 -15912.062,E2 -15912.062} C_VEL
LIN {X 0,Y 306.143,Z 458.425,A -85,B 0,C 180,E1 -15914.616,E2 -15914.616} C_VEL
LIN {X 0,Y 304.969,Z 464.379,A -85,B 0,C 180,E1 -15917.354,E2 -15917.354} C_VEL
LIN {X 0,Y 304.26,Z 467.844,A -85,B 0,C 180,E1 -15919.352,E2 -15919.352} C_VEL
LIN {X 0,Y 303.774,Z 471.343,A -85,B 0,C 180,E1 -15922.021,E2 -15922.021} C_VEL
LIN {X 0,Y 303.595,Z 473.66,A -85,B 0,C 180,E1 -15924.687,E2 -15924.687} C_VEL
LIN {X 0,Y 303.587,Z 474.838,A -85,B 0,C 180,E1 -15927.347,E2 -15927.347} C_VEL
LIN {X 0,Y 303.602,Z 474.86,A -85,B 0,C 180,E1 -15930.001,E2 -15930.001} C_VEL
LIN {X 0,Y 303.595,Z 473.679,A -85,B 0,C 180,E1 -15932.654,E2 -15932.654} C_VEL
LIN {X 0,Y 303.623,Z 471.064,A -85,B 0,C 180,E1 -15935.545,E2 -15935.545} C_VEL
LIN {X 0,Y 303.801,Z 467.723,A -85,B 0,C 180,E1 -15937.979,E2 -15937.979} C_VEL
LIN {X 0,Y 304.116,Z 462.785,A -85,B 0,C 180,E1 -15940.655,E2 -15940.655} C_VEL
LIN {X 0,Y 304.938,Z 456.382,A -85,B 0,C 180,E1 -15943.326,E2 -15943.326} C_VEL
LIN {X 0,Y 306.134,Z 448.319,A -85,B 0,C 180,E1 -15945.992,E2 -15945.992} C_VEL
LIN {X 0,Y 307.575,Z 439.705,A -85,B 0,C 180,E1 -15948.312,E2 -15948.312} C_VEL
LIN {X 0,Y 309.255,Z 430.969,A -85,B 0,C 180,E1 -15950.278,E2 -15950.278} C_VEL
LIN {X 0,Y 311.165,Z 419.797,A -85,B 0,C 180,E1 -15952.377,E2 -15952.377} C_VEL
LIN {X 0,Y 313.315,Z 408.211,A -85,B 0,C 180,E1 -15954.166,E2 -15954.166} C_VEL
LIN {X 0,Y 315.348,Z 395.755,A -85,B 0,C 180,E1 -15955.76,E2 -15955.76} C_VEL
LIN {X 0,Y 317.318,Z 383.804,A -85,B 0,C 180,E1 -15957.004,E2 -15957.004} C_VEL
LIN {X 0,Y 319.142,Z 370.451,A -85,B 0,C 180,E1 -15958.146,E2 -15958.146} C_VEL
LIN {X 0,Y 320.687,Z 356.415,A -85,B 0,C 180,E1 -15959.095,E2 -15959.095} C_VEL
LIN {X 0,Y 322.22,Z 341.212,A -85,B 0,C 180,E1 -15959.84,E2 -15959.84} C_VEL
LIN {X 0,Y 323.157,Z 325.203,A -85,B 0,C 180,E1 -15960.375,E2 -15960.375} C_VEL
LIN {X 0,Y 326.714,Z 214.794,A -85,B 0,C 180,E1 -15962.818,E2 -15962.818} C_VEL
LIN {X 0,Y 323.522,Z 195.882,A -85,B 0,C 180,E1 -15963.597,E2 -15963.597} C_VEL
LIN {X 0,Y 314.439,Z 174.008,A -85,B 0,C 180,E1 -15965.079,E2 -15965.079} C_VEL
LIN {X 0,Y 309.272,Z 162.47,A -85,B 0,C 180,E1 -15965.967,E2 -15965.967} C_VEL
LIN {X 0,Y 306.29,Z 151.066,A -85,B 0,C 180,E1 -15969.15,E2 -15969.15} C_VEL
LIN {X 0,Y 305.476,Z 148.059,A -85,B 0,C 180,E1 -15970.054,E2 -15970.054} C_VEL
LIN {X 0,Y 305.427,Z 148.069,A -85,B 0,C 180,E1 -15973.656,E2 -15973.656} C_VEL
LIN {X 0,Y 305.457,Z 148.065,A -85,B 0,C 180,E1 -15977.415,E2 -15977.415} C_VEL
LIN {X 0,Y 305.469,Z 148.051,A -85,B 0,C 180,E1 -15981.597,E2 -15981.597} C_VEL
LIN {X 0,Y 305.464,Z 148.057,A -85,B 0,C 180,E1 -15984.888,E2 -15984.888} C_VEL
LIN {X 0,Y 305.444,Z 148.06,A -85,B 0,C 180,E1 -15988.359,E2 -15988.359} C_VEL
LIN {X 0,Y 305.478,Z 148.039,A -85,B 0,C 180,E1 -15991.11,E2 -15991.11} C_VEL
LIN {X 0,Y 305.503,Z 148.042,A -85,B 0,C 180,E1 -15994.082,E2 -15994.082} C_VEL
LIN {X 0,Y 305.479,Z 148.049,A -85,B 0,C 180,E1 -15998.402,E2 -15998.402} C_VEL
LIN {X 0,Y 305.55,Z 148.047,A -85,B 0,C 180,E1 -16001.216,E2 -16001.216} C_VEL
LIN {X 0,Y 305.63,Z 148.039,A -85,B 0,C 180,E1 -16005.349,E2 -16005.349} C_VEL
LIN {X 0,Y 305.629,Z 148.038,A -85,B 0,C 180,E1 -16009.4,E2 -16009.4} C_VEL
LIN {X 0,Y 305.75,Z 148.019,A -85,B 0,C 180,E1 -16012.073,E2 -16012.073} C_VEL
LIN {X 0,Y 305.662,Z 148.035,A -85,B 0,C 180,E1 -16014.724,E2 -16014.724} C_VEL
LIN {X 0,Y 305.939,Z 147.969,A -85,B 0,C 180,E1 -16018.684,E2 -16018.684} C_VEL
LIN {X 0,Y 305.938,Z 147.982,A -85,B 0,C 180,E1 -16021.317,E2 -16021.317} C_VEL
LIN {X 0,Y 305.79,Z 148.008,A -85,B 0,C 180,E1 -16026.599,E2 -16026.599} C_VEL
LIN {X 0,Y 305.698,Z 147.994,A -85,B 0,C 180,E1 -16029.261,E2 -16029.261} C_VEL
LIN {X 0,Y 305.558,Z 148.042,A -85,B 0,C 180,E1 -16033.298,E2 -16033.298} C_VEL
LIN {X 0,Y 305.493,Z 148.05,A -85,B 0,C 180,E1 -16036.026,E2 -16036.026} C_VEL
LIN {X 0,Y 305.481,Z 148.058,A -85,B 0,C 180,E1 -16039.392,E2 -16039.392} C_VEL
LIN {X 0,Y 305.46,Z 148.054,A -85,B 0,C 180,E1 -16043.026,E2 -16043.026} C_VEL
LIN {X 0,Y 305.455,Z 148.055,A -85,B 0,C 180,E1 -16046.19,E2 -16046.19} C_VEL
LIN {X 0,Y 305.426,Z 148.032,A -85,B 0,C 180,E1 -16049.025,E2 -16049.025} C_VEL
LIN {X 0,Y 305.441,Z 148.054,A -85,B 0,C 180,E1 -16051.953,E2 -16051.953} C_VEL
LIN {X 0,Y 305.466,Z 148.056,A -85,B 0,C 180,E1 -16055.114,E2 -16055.114} C_VEL
LIN {X 0,Y 305.438,Z 148.033,A -85,B 0,C 180,E1 -16058.525,E2 -16058.525} C_VEL
LIN {X 0,Y 305.44,Z 148.064,A -85,B 0,C 180,E1 -16062.582,E2 -16062.582} C_VEL
